Yaskawa INFORM job: X2_8B-21B(90,180)_REV_O.JBI

/JOB
//NAME X2_8B-21B(90,180)_REV_O
///FOLDERNAME X2
//POS
///NPOS 1154,1154,1154,53,0,0
///TOOL 0
///POSTYPE PULSE
///PULSE
C00000=-1415,-134459,-133802,-1969,12985,79332
C00001=-87080,-112473,-103627,-41798,51237,70410
C00002=-91681,-107347,-99471,-39221,49165,68848
C00003=-93439,-105106,-97054,-38371,48113,68361
C00004=-93441,-104864,-95967,-38672,47682,68565
C00005=-93504,-104969,-96260,-38564,47753,68495
C00006=-95585,-102642,-95415,-36914,47385,67494
C00007=-93504,-104969,-96260,-38564,47753,68495
C00008=-87147,-112175,-102116,-42180,50619,70689
C00009=-87145,-119394,-106475,-25944,48524,38750
C00010=-91166,-110510,-101811,-22693,48895,36705
C00011=-92650,-107060,-99920,-21494,49065,35962
C00012=-94767,-104655,-99060,-19829,49198,34943
C00013=-94484,-105085,-99259,-20052,49173,35080
C00014=-93721,-102513,-96995,-20598,49294,35408
C00015=-94484,-105085,-99259,-20052,49173,35080
C00016=-89209,-117497,-105909,-24366,48468,37757
C00017=-93166,-113214,-115710,-1969,57926,79332
C00018=-122366,-117496,-112293,16338,56235,67679
C00019=-123456,-103417,-106445,16337,59944,67813
C00020=-123456,-103539,-105172,16474,59132,67689
C00021=-123456,-103531,-105272,16463,59195,67698
C00022=-123128,-98284,-103303,16044,60561,68033
C00023=-123156,-99911,-105489,15984,61057,68095
C00024=-93710,-106990,-108704,-1652,56802,79139
C00025=-93766,-106412,-107148,-1629,56140,79127
C00026=-93768,-106433,-106329,-1638,55626,79135
C00027=-93918,-105383,-106173,-1535,56065,79069
C00028=-94164,-101296,-104676,-1361,57240,78956
C00029=-93895,-105502,-106499,-1547,56205,79076
C00030=-93151,-113316,-114305,-1998,57010,79354
C00031=-81072,-99391,-111155,-4750,63110,78553
C00032=-81984,-95120,-104767,-4287,61328,78293
C00033=-82103,-94682,-103397,-4241,60705,78273
C00034=-82106,-94924,-102383,-4271,59960,78300
C00035=-82089,-94934,-102578,-4276,60076,78302
C00036=-82803,-90374,-100753,-3806,61258,77993
C00037=-82089,-94934,-102578,-4276,60076,78302
C00038=-81057,-100006,-109908,-4804,62030,78604
C00039=-94004,-119945,-107122,49530,42714,48164
C00040=-93972,-116281,-97047,53343,39935,45878
C00041=-92833,-103149,-88492,51302,40218,47068
C00042=-93174,-100930,-87132,51219,40604,47120
C00043=-93174,-100493,-85792,51770,40220,46795
C00044=-93174,-101015,-87399,51095,40684,47186
C00045=-92955,-97894,-86230,50180,41136,47726
C00046=-93303,-100448,-87190,51023,40860,47230
C00047=-98055,-98607,-86499,53149,43882,46024
C00048=-96642,-96320,-85623,51883,43475,46780
C00049=-95342,-96864,-85830,51299,42647,47109
C00050=-97130,-98187,-86063,52744,43317,46271
C00051=-114545,-105110,-100746,39625,57097,48369
C00052=-113947,-102413,-97570,39574,56382,48359
C00053=-113947,-102278,-96691,39772,56015,48196
C00054=-113346,-99976,-96570,39024,56612,48763
C00055=-112899,-98120,-95866,38597,56823,49078
C00056=-114020,-99555,-96940,39169,57262,48705
C00057=-56302,-84822,-83054,-58022,66572,84014
C00058=-58361,-85953,-83540,-57558,65172,83717
C00059=-56302,-84822,-83054,-58022,66572,84014
C00060=-50122,-85714,-86741,-59061,71306,84454
C00061=-54195,-101901,-111197,-24063,62262,77343
C00062=-67243,-111926,-101536,21450,29925,69540
C00063=-66442,-101704,-94400,19916,30532,70304
C00064=-66308,-99858,-92576,19846,30336,70336
C00065=-66311,-99589,-91307,20230,29731,70137
C00066=-66308,-99960,-93112,19687,30597,70418
C00067=-70591,-100617,-92786,25268,31264,67678
C00068=-70591,-100325,-91437,25755,30647,67424
C00069=-68222,-99738,-91214,22742,30105,68906
C00070=-70591,-100606,-92729,25289,31242,67667
C00071=-66097,-110297,-96199,21577,27345,69446
C00072=-65719,-107666,-92844,21562,26575,69447
C00073=-65848,-106528,-92445,21497,26927,69482
C00074=-65365,-110699,-93884,21743,25627,69354
C00075=-67243,-111926,-101536,21450,29925,69540
C00076=-68963,-41843,-96211,-398,96948,-48811
C00077=-76932,-51697,-92360,2602,89609,-51106
C00078=-71886,-45093,-85416,705,88639,-49643
C00079=-71886,-45937,-84760,705,87803,-49648
C00080=-71886,-44632,-85753,705,89084,-49641
C00081=-68776,-90352,-95136,-4313,51281,-47645
C00082=-68803,-86754,-93636,-4241,52203,-47695
C00083=-68762,-92243,-95906,-4353,50785,-47617
C00084=-77446,-64871,-91176,8832,74282,-49527
C00085=-75907,-64612,-91046,8095,74185,-49034
C00086=-78150,-64967,-91224,9168,74335,-49752
C00087=-78150,-57569,-97635,8943,81990,-49191
C00088=-68963,-41843,-96211,-398,96948,-48811
C00089=-67385,-42511,-92598,-992,94393,-48367
C00090=-66773,-44328,-90253,-1220,92024,-48175
C00091=-66900,-44765,-89647,-1171,91425,-48205
C00092=-66773,-43962,-90441,-1221,92327,-48178
C00093=-69817,-49291,-93527,-72,91467,-49038
C00094=-102407,-61387,-79216,48101,75803,-74984
C00095=-99741,-62884,-79905,47237,74215,-74494
C00096=-102407,-61387,-79216,48101,75803,-74984
C00097=-71396,-101707,-96198,105,39560,-49678
C00098=-71544,-99303,-95354,247,40276,-49753
C00099=-71126,-105930,-97636,-165,38275,-49535
C00100=-74447,-120283,-111838,3099,39699,-51260
C00101=-57750,-84762,-113304,-22338,79933,-80646
C00102=-38298,-117376,-123136,-35520,84192,-83183
C00103=-31003,-114098,-105660,-45955,85390,-81321
C00104=-32496,-116782,-107403,-45795,84408,-81579
C00105=-34116,-118987,-108120,-45640,83088,-81742
C00106=-33779,-118873,-108083,-45678,83285,-81673
C00107=-33779,-118389,-106291,-45736,82677,-81394
C00108=-33116,-116007,-107005,-45711,84199,-81779
C00109=-43122,-77390,-91933,-43525,86904,-87571
C00110=-44353,-78017,-92219,-43231,86215,-87819
C00111=-45440,-79271,-92786,-42975,85486,-87990
C00112=-45102,-79332,-92813,-43057,85636,-87902
C00113=-45102,-79709,-91490,-43095,84888,-87585
C00114=-41853,-68825,-87871,-43817,88900,-87868
C00115=-48095,-31712,-66541,-47290,99218,-86920
C00116=-48762,-33638,-67810,-47108,98755,-86994
C00117=-49503,-35735,-69173,-46902,98237,-87073
C00118=-49389,-35416,-68966,-46933,98317,-87062
C00119=-49389,-36060,-68028,-46814,97684,-86756
C00120=-48487,-32850,-67294,-47182,98948,-86964
C00121=-45126,-25671,-76382,-49967,106798,-89554
C00122=-48508,-32956,-85951,-38791,109748,-85822
C00123=-73491,-115415,-129730,-12591,84406,-82629
C00124=-68604,-111632,-124361,34026,103601,-55041
C00125=-52690,-105642,-114364,31889,95098,-51390
C00126=-50963,-109289,-114635,31553,93010,-51314
C00127=-50968,-109442,-114037,31534,92627,-51422
C00128=-50963,-109237,-114816,31559,93129,-51281
C00129=-54701,-101748,-112541,32228,96580,-51739
C00130=-54580,-102143,-110625,32107,95358,-52042
C00131=-52710,-105778,-111943,31798,93771,-51772
C00132=-54580,-102143,-110625,32107,95358,-52042
C00133=-53574,-106836,-112314,31893,93817,-52092
C00134=-52008,-102475,-110737,31756,94333,-51344
C00135=-53574,-106836,-112314,31893,93817,-52092
C00136=-61074,-96775,-114868,33501,102293,-52496
C00137=-149084,-102156,-129577,22032,95315,-42360
C00138=-128569,-114069,-129208,14930,94899,-36248
C00139=-124702,-111484,-125119,14131,93099,-35189
C00140=-117407,-110681,-122838,12596,90996,-33018
C00141=-117407,-111232,-122133,12590,90297,-33088
C00142=-117407,-111153,-122240,12590,90402,-33077
C00143=-117516,-104258,-119840,12640,92435,-32906
C00144=-117407,-111153,-122240,12590,90402,-33077
C00145=-137517,-133828,-121685,31184,78220,-41365
C00146=-133868,-135584,-122192,30484,76378,-40422
C00147=-116503,-109521,-121739,12400,90787,-32743
C00148=-117639,-111560,-122305,12792,90174,-33159
C00149=-129920,-104375,-121589,15367,95339,-36612
C00150=-129920,-105073,-120932,15342,94602,-36705
C00151=-129920,-105823,-120129,15315,93754,-36812
C00152=-129920,-105714,-120250,15319,93879,-36798
C00153=-129568,-97895,-117405,15323,96007,-36416
C00154=-129817,-102709,-120162,15344,95301,-36587
C00155=-121595,-114825,-128025,13496,92670,-34216
C00156=-122629,-107467,-122921,17549,92277,-31147
C00157=-121348,-106187,-119304,17235,90519,-30969
C00158=-121348,-106897,-118296,17228,89578,-31103
C00159=-121348,-106810,-118429,17228,89701,-31085
C00160=-121327,-99353,-115727,17255,91773,-30786
C00161=-121340,-102686,-118046,17252,91502,-30828
C00162=-123984,-121300,-124584,22039,85383,-28695
C00163=-118596,-113071,-118409,20758,84424,-26972
C00164=-117828,-112575,-117002,20585,83663,-26833
C00165=-117596,-112721,-116348,20543,83158,-26838
C00166=-117643,-112201,-116474,20543,83493,-26797
C00167=-117846,-106122,-114344,20549,85245,-26570
C00168=-117643,-112201,-116474,20543,83493,-26797
C00169=-125192,-113488,-115877,22341,84450,-29296
C00170=-124919,-116220,-115928,22323,83104,-29449
C00171=-122352,-116155,-116251,21738,82647,-28614
C00172=-124919,-116220,-115928,22323,83104,-29449
C00173=-123984,-121300,-124584,22039,85383,-28695
C00174=-86442,-134681,-133724,-19248,79211,-32552
C00175=-86002,-121949,-124889,-19319,80358,-32581
C00176=-83173,-118115,-122503,-20102,81494,-31775
C00177=-83173,-118355,-121819,-20128,80982,-31690
C00178=-83173,-118313,-121945,-20123,81076,-31705
C00179=-84570,-111270,-119601,-19642,82802,-32476
C00180=-84061,-113318,-121554,-19798,83063,-32340
C00181=-99760,-154859,-112577,-64842,65446,-34340
C00182=-105860,-151698,-110493,-64559,61681,-35508
C00183=-106986,-150846,-109245,-64674,60811,-35545
C00184=-106922,-150967,-109400,-64661,60866,-35548
C00185=-107498,-146229,-108289,-63778,61296,-36463
C00186=-107239,-150553,-110467,-64221,61056,-36009
C00187=-103039,-154525,-109995,-65437,62710,-34223
C00188=-103986,-153521,-108660,-65576,61968,-34235
C00189=-103986,-153752,-108910,-65558,61982,-34250
C00190=-104831,-148338,-107690,-64592,62341,-35332
C00191=-104831,-154990,-115289,-64019,62915,-35911
C00192=-86002,-121949,-124889,-19319,80358,-32581
C00193=-89184,-120947,-124012,-18384,79622,-33578
C00194=-89184,-121311,-122777,-18433,78722,-33443
C00195=-89184,-121280,-122900,-18428,78809,-33455
C00196=-90163,-115208,-120930,-18039,80412,-34039
C00197=-89061,-121712,-124317,-18429,79452,-33511
C00198=-95932,-170316,-132534,-19010,48950,-33315
C00199=-95449,-171774,-131482,-19685,47748,-32835
C00200=-93413,-168537,-129826,-20545,48851,-32116
C00201=-93413,-168812,-130071,-20542,48860,-32116
C00202=-94803,-159418,-127836,-18887,51784,-33360
C00203=-94151,-164650,-129663,-19626,50457,-32799
C00204=-96358,-174071,-130551,-19748,45875,-32859
C00205=-95061,-171972,-129445,-20316,46563,-32383
C00206=-95061,-172212,-129646,-20316,46563,-32383
C00207=-96259,-163989,-127758,-18767,49173,-33508
C00208=-95716,-170264,-130833,-19432,48038,-33021
C00209=-120611,-122953,-119681,21560,80854,-22535
C00210=-120610,-122943,-118608,21593,80243,-22645
C00211=-120610,-122853,-116921,21650,79318,-22813
C00212=-120610,-122881,-117271,21638,79506,-22779
C00213=-120610,-122878,-117279,21638,79511,-22778
C00214=-120610,-122881,-117271,21638,79506,-22779
C00215=-120610,-122873,-117198,21640,79468,-22785
C00216=-120610,-122853,-117190,21640,79473,-22785
C00217=-120610,-122873,-117198,21640,79468,-22785
C00218=-120611,-122910,-120952,21522,81605,-22399
C00219=-86002,-120340,-127953,-19212,82925,-32989
C00220=-83173,-118115,-122503,-20102,81494,-31775
C00221=-83173,-118354,-121819,-20128,80983,-31690
C00222=-83173,-118313,-121945,-20123,81076,-31705
C00223=-84570,-111270,-119601,-19642,82802,-32476
C00224=-84061,-113318,-121554,-19798,83063,-32340
C00225=-99760,-154859,-112577,-64842,65446,-34340
C00226=-105859,-151698,-110493,-64559,61681,-35508
C00227=-106987,-150846,-109245,-64674,60811,-35545
C00228=-106922,-150967,-109400,-64660,60866,-35548
C00229=-107498,-146229,-108289,-63777,61296,-36463
C00230=-107240,-150553,-110467,-64221,61056,-36009
C00231=-103039,-154525,-109995,-65437,62710,-34223
C00232=-103986,-153521,-108660,-65576,61968,-34235
C00233=-103986,-153752,-108910,-65558,61982,-34249
C00234=-104831,-148338,-107690,-64592,62341,-35332
C00235=-104831,-154990,-115290,-64019,62915,-35911
C00236=-86002,-121950,-124889,-19319,80357,-32581
C00237=-89184,-120947,-124012,-18384,79622,-33578
C00238=-89184,-121311,-122777,-18433,78722,-33443
C00239=-89184,-121280,-122899,-18429,78809,-33455
C00240=-90163,-115207,-120930,-18039,80412,-34039
C00241=-89061,-121712,-124317,-18429,79452,-33511
C00242=-95932,-170316,-132534,-19010,48950,-33315
C00243=-95449,-171774,-131482,-19685,47748,-32835
C00244=-93413,-168536,-129826,-20544,48851,-32117
C00245=-93413,-168811,-130070,-20542,48860,-32116
C00246=-94803,-159417,-127836,-18887,51784,-33360
C00247=-94151,-164650,-129664,-19626,50457,-32799
C00248=-96358,-174071,-130551,-19748,45875,-32859
C00249=-95060,-171973,-129446,-20316,46563,-32383
C00250=-95061,-172212,-129646,-20316,46563,-32383
C00251=-96259,-163989,-127758,-18767,49173,-33508
C00252=-95716,-170264,-130834,-19432,48038,-33021
C00253=-120612,-120891,-127143,3106,87300,-4415
C00254=-120611,-122177,-124352,3111,84925,-4474
C00255=-120611,-122645,-122467,3116,83527,-4507
C00256=-120611,-122779,-121606,3119,82929,-4523
C00257=-120611,-122697,-122159,3117,83311,-4513
C00258=-120611,-122692,-122166,3117,83318,-4513
C00259=-120611,-122697,-122159,3117,83311,-4513
C00260=-120611,-121412,-126223,3107,86468,-4436
C00261=-120611,-118807,-129728,3107,89959,-4350
C00262=-120605,-132560,-136700,3104,87187,-4416
C00263=-53188,-122658,-121398,34453,103181,-41719
C00264=-53187,-122644,-116623,34032,100735,-42492
C00265=-53184,-122447,-115007,33919,99986,-42724
C00266=-53180,-122268,-113886,33849,99484,-42877
C00267=-53186,-122531,-115629,33961,100272,-42636
C00268=-53233,-122033,-113114,32057,113501,-44659
C00269=-53229,-122037,-113108,32057,113495,-44659
C00270=-53233,-122033,-113114,32057,113501,-44659
C00271=-53127,-122157,-112856,34567,84618,-41563
C00272=-53132,-122146,-112848,34568,84621,-41564
C00273=-53127,-122157,-112856,34567,84618,-41563
C00274=-53124,-122720,-116247,34514,86111,-41098
C00275=-61684,-126457,-131749,21672,103686,-55019
C00276=-68676,-133744,-131015,10578,108811,-68614
C00277=-80160,-118182,-130261,-41,125141,-81817
C00278=-80187,-122370,-123619,-70,118933,-81856
C00279=-80183,-122639,-122398,-68,118043,-81854
C00280=-80181,-122756,-121636,-67,117515,-81853
C00281=-80184,-122603,-122588,-68,118179,-81854
C00282=-80182,-122615,-122584,-67,118170,-81853
C00283=-80184,-122603,-122588,-68,118179,-81854
C00284=-80200,-121154,-126606,-75,121396,-81862
C00285=-109164,-117358,-132635,-7350,119146,-48306
C00286=-144183,-119511,-130571,-15498,107286,-7245
C00287=-197934,-122815,-127402,-28006,89082,55776
C00288=-202772,-123889,-124791,-27048,85608,54814
C00289=-204705,-124106,-122314,-26692,83530,54575
C00290=-204705,-124189,-120905,-26732,82711,54762
C00291=-205113,-122699,-120601,-26621,83104,54520
C00292=-208506,-122040,-120392,-25870,82241,53457
C00293=-204510,-125657,-121990,-26775,82699,54838
C00294=-204510,-125393,-124777,-26704,84359,54459
C00295=-217123,-144581,-130617,-26990,80795,43719
C00296=-208514,-157553,-136215,-22784,79668,13108
C00297=-208134,-153606,-128050,-23049,77001,13769
C00298=-209226,-147410,-126429,-22728,78719,13024
C00299=-208514,-151468,-127497,-22936,77598,13510
C00300=-218941,-132344,-125800,-20692,83017,8703
C00301=-218940,-132255,-124809,-20728,82492,8794
C00302=-218940,-132304,-125288,-20718,82746,8752
C00303=-219615,-126196,-123449,-20528,84462,8218
C00304=-218940,-132304,-125288,-20718,82746,8752
C00305=-200084,-117243,-114643,-37064,92847,22860
C00306=-201812,-115748,-114150,-36926,92488,22266
C00307=-218940,-132304,-125288,-20718,82746,8752
C00308=-203904,-153254,-131986,6783,67239,16317
C00309=-203904,-152472,-130784,6798,66902,16298
C00310=-203904,-152823,-131321,6790,67052,16308
C00311=-205098,-146177,-129554,7075,69466,16016
C00312=-203904,-152823,-131321,6790,67052,16308
C00313=-223566,-125183,-123361,20045,84784,-13848
C00314=-220870,-123350,-122791,19484,84702,-12913
C00315=-222373,-123821,-125769,19771,86556,-13139
C00316=-208514,-151468,-127497,-22936,77598,13510
C00317=-208514,-156517,-134755,-22805,79329,13174
C00318=-197934,-122815,-127402,-28006,89082,55776
C00319=-202772,-123889,-124791,-27048,85608,54814
C00320=-204705,-124106,-122314,-26692,83530,54575
C00321=-204705,-124189,-120905,-26732,82711,54762
C00322=-205113,-122699,-120601,-26621,83104,54520
C00323=-208506,-122040,-120392,-25870,82241,53457
C00324=-204510,-125657,-121990,-26775,82699,54838
C00325=-204510,-125393,-124777,-26704,84359,54459
C00326=-217123,-144581,-130617,-26990,80795,43719
C00327=-216657,-144339,-132121,-20327,83655,24427
C00328=-208514,-151468,-127497,-22936,77598,13510
C00329=-209226,-147410,-126429,-22728,78719,13024
C00330=-208514,-151468,-127497,-22936,77598,13510
C00331=-208514,-156517,-134755,-22805,79329,13174
C00332=-187736,-116553,-120968,-36188,98329,31010
C00333=-144869,-104708,-130913,697,92502,-12445
C00334=-97478,-100538,-119508,25976,122096,-72949
C00335=-94415,-115583,-120723,24602,114867,-73486
C00336=-94145,-116737,-119872,24403,113768,-73630
C00337=-94090,-116915,-118863,24267,113100,-73760
C00338=-94227,-118887,-121662,24392,113788,-73658
C00339=-94618,-126072,-123928,23885,111795,-74261
C00340=-93811,-121058,-122280,24303,112998,-73673
C00341=-123165,-134656,-120887,30393,109989,-65140
C00342=-122877,-135920,-118822,30065,108215,-65520
C00343=-120918,-135771,-118381,30417,107339,-64954
C00344=-122877,-135920,-118822,30065,108215,-65520
C00345=-123434,-129548,-123417,31323,113703,-64157
C00346=-83798,-143971,-127552,34208,94145,-53659
C00347=-12921,-128304,-123041,22509,73309,-31557
C00348=-1276,-141206,-132907,9958,77401,-32714
C00349=458,-143834,-132257,9551,75469,-32266
C00350=455,-143428,-130846,9594,74819,-32314
C00351=455,-143488,-131041,9589,74909,-32308
C00352=3648,-143226,-130969,8703,74636,-31209
C00353=1152,-143828,-132318,9375,75428,-32023
C00354=8026,-156372,-135202,7630,70086,-29960
C00355=9901,-151141,-133831,7007,71746,-29188
C00356=9901,-150525,-132660,7023,71345,-29214
C00357=9901,-150622,-132845,7021,71407,-29209
C00358=13681,-148784,-132355,5888,71743,-27846
C00359=12497,-150457,-134690,6220,72408,-28233
C00360=-126606,-101457,-128935,16844,101795,-36174
C00361=-152779,-135138,-131563,2515,76140,-19155
C00362=-150820,-122490,-124749,1875,78392,-18455
C00363=-150097,-118368,-121531,1645,78513,-18212
C00364=-150095,-118599,-120646,1648,77850,-18220
C00365=-147666,-112236,-119185,871,80184,-17389
C00366=-146670,-110099,-118456,556,80825,-17059
C00367=-148658,-114325,-119887,1186,79554,-17722
C00368=-87079,-91764,-103818,-42328,107533,9448
C00369=-87027,-91004,-101788,-42122,106912,9740
C00370=-89264,-90509,-101588,-42089,105978,9119
C00371=-87027,-91004,-101788,-42122,106912,9740
C00372=-87391,-90282,-107909,-43186,109836,8282
C00373=-92115,-87061,-118989,-19004,94950,-3823
C00374=-109005,-100727,-117090,5533,93286,-3886
C00375=-109005,-102030,-115406,5521,91587,-3960
C00376=-109005,-101552,-116078,5524,92244,-3931
C00377=-107643,-92243,-112443,5266,94693,-3390
C00378=-109005,-99994,-117863,5541,94135,-3847
C00379=-92115,-87061,-118989,-19004,94950,-3823
C00380=-78975,-130870,-123203,19746,71053,-12291
C00381=-74317,-97013,-111518,17407,83606,-9286
C00382=-74211,-95430,-110119,17377,83539,-9259
C00383=-74211,-95892,-109317,17397,82840,-9358
C00384=-75305,-113551,-114600,17838,69768,-10493
C00385=-78326,-111051,-111958,19079,70114,-11550
C00386=-78379,-106110,-110225,18937,71523,-11339
C00387=-78263,-116865,-113913,19272,68408,-11810
C00388=-85880,-113569,-112821,22054,71256,-14152
C00389=-85920,-114580,-110580,22309,69503,-14507
C00390=-82054,-114988,-110714,20879,68380,-13249
C00391=-85920,-114580,-110580,22309,69503,-14507
C00392=-78975,-130870,-123203,19746,67177,-12291
C00393=-159950,-115131,-126913,-23322,109234,64770
C00394=-163413,-124246,-126581,-22686,103792,64589
C00395=-164859,-127477,-125491,-22457,101245,64551
C00396=-164857,-127553,-124648,-22406,100728,64651
C00397=-164862,-127370,-126252,-22506,101730,64457
C00398=-158275,-145382,-129341,-21795,96649,67831
C00399=-159759,-153222,-131425,-21726,93697,67826
C00400=-158275,-145382,-129341,-21795,96649,67831
C00401=-157577,-144643,-126617,-21696,95625,68274
C00402=-160219,-140867,-125578,-21868,96138,67212
C00403=-157577,-144643,-126617,-21696,95625,68274
C00404=-152631,-134238,-128202,-21932,102817,68768
C00405=-146941,-123801,-133763,-3444,102850,52685
C00406=-136178,-116173,-124987,31736,84906,22811
C00407=-134413,-106132,-117362,31242,84680,23412
C00408=-134231,-105594,-115694,31219,83968,23286
C00409=-134230,-105863,-115134,31239,83552,23172
C00410=-134007,-104199,-114803,31151,84035,23389
C00411=-133473,-100630,-113499,30965,84737,23780
C00412=-134315,-106237,-115533,31260,83629,23161
C00413=-136272,-117460,-124003,31807,83855,22481
C00414=-136226,-116324,-125056,31750,84893,22789
C00415=-134474,-106353,-117504,31259,84679,23389
C00416=-134275,-105758,-115681,31235,83904,23252
C00417=-134274,-105987,-115198,31252,83547,23154
C00418=-134027,-104733,-115029,31162,83924,23350
C00419=-133465,-100971,-113658,30966,84667,23763
C00420=-134308,-106598,-115693,31262,83551,23142
C00421=-178993,-121773,-123174,38769,99022,10273
C00422=-175539,-115427,-119854,38657,98481,11541
C00423=-175539,-115857,-118311,38525,97555,11203
C00424=-175539,-115829,-118427,38535,97623,11227
C00425=-173168,-111114,-116839,38478,97741,12267
C00426=-174072,-113112,-119760,38657,98741,12252
C00427=-136269,-117902,-124178,31812,83752,22453
C00428=-139753,-124875,-130430,383,75663,-26245
C00429=-143223,-157944,-133481,-5653,58679,-38405
C00430=-140983,-144085,-126452,-6488,61628,-37698
C00431=-140148,-138933,-122655,-6835,62006,-37402
C00432=-140147,-138616,-121921,-6853,61719,-37384
C00433=-140691,-136506,-121897,-6553,62737,-37651
C00434=-138669,-131542,-120459,-7325,64564,-37004
C00435=-140691,-136506,-121897,-6553,62737,-37651
C00436=-145148,-139028,-124584,-4588,62787,-39337
C00437=-159973,-92454,-110285,14523,90938,-48717
C00438=-158765,-97223,-112137,14224,89465,-48492
C00439=-159973,-92454,-110285,14523,90938,-48717
C00440=-164681,-91509,-114703,15696,94847,-49769
C00441=-142525,-105883,-132766,-7713,103357,-60336
C00442=-90751,-115691,-121566,-36045,104861,-61043
C00443=-92920,-122587,-117773,-35137,99152,-60047
C00444=-93124,-123070,-117553,-35091,98753,-60003
C00445=-93124,-123008,-116878,-35050,98435,-59900
C00446=-93160,-123063,-117190,-35068,98555,-59953
C00447=-95752,-125144,-117838,-34977,96947,-60505
C00448=-93160,-123063,-117190,-35068,98555,-59953
C00449=-92038,-109836,-114685,-38536,89453,-57060
C00450=-86810,-100893,-104585,-47463,92019,-56975
C00451=-88449,-102594,-103600,-47188,90148,-56855
C00452=-88449,-102618,-102426,-47172,89639,-56610
C00453=-88449,-102603,-103366,-47184,90046,-56806
C00454=-85133,-99388,-102162,-47637,92393,-56350
C00455=-85168,-99488,-101153,-47595,91912,-56132
C00456=-86978,-101259,-101820,-47360,90627,-56378
C00457=-84037,-98201,-102123,-47804,93363,-56297
C00458=-108771,-112096,-123986,-16313,85813,-59347
C00459=-109769,-112695,-132242,-3132,99947,-61138
C00460=-127404,-127157,-120795,27540,73197,-60883
C00461=-120526,-123085,-115007,25540,69700,-59025
C00462=-119461,-122312,-114032,25210,69192,-58723
C00463=-119461,-122116,-113003,25293,68708,-58832
C00464=-119461,-122312,-114032,25210,69192,-58723
C00465=-94655,-112249,-115827,-1041,75214,-51009
C00466=-93364,-111129,-115444,-1499,75574,-50577
C00467=-121213,-123445,-114215,25873,69302,-59387
C00468=-127714,-127278,-119628,27738,72603,-61150
C00469=-140848,-129628,-128054,17424,84805,-27418
C00470=-127903,-106251,-120637,17388,91568,-15860
C00471=-124887,-98361,-114445,16717,91208,-14907
C00472=-124532,-94860,-112080,16625,91471,-14753
C00473=-117832,-103976,-115449,15062,87719,-13014
C00474=-118209,-109888,-118953,15141,86934,-13233
C00475=-120968,-118649,-124805,15800,86569,-14208
C00476=-112726,-101228,-128594,1890,90279,15897
C00477=-102865,-105549,-130121,-1361,88970,18873
C00478=-85416,-143080,-122146,-23399,58401,32529
C00479=-89847,-131888,-116792,-20882,59491,30436
C00480=-92125,-126361,-114096,-19602,60042,29398
C00481=-92108,-126361,-114086,-19611,60041,29405
C00482=-94963,-119193,-112807,-13876,65309,25883
C00483=-99230,-109273,-111594,-7832,72910,21884
C00484=-97558,-114678,-114533,-8498,72116,22521
C00485=-94805,-124749,-120489,-9597,70928,23580
C00486=-89899,-115674,-129227,-15589,81503,27304
C00487=-94000,-113154,-130859,1035,116659,-75004
C00488=-93721,-118000,-129934,5060,122177,-74127
C00489=-93715,-120352,-127357,4900,119392,-74256
C00490=-95346,-120435,-125547,4467,118331,-74923
C00491=-87734,-123112,-126247,6115,116903,-72103
C00492=-93725,-120284,-127319,4898,119404,-74259
C00493=-93731,-117931,-129895,5059,122189,-74130
C00494=-92605,-107385,-114202,-42080,118626,-78084
C00495=-94957,-117308,-114744,-40643,113912,-77125
C00496=-96859,-119647,-113709,-40343,111617,-77062
C00497=-96820,-119688,-113698,-40330,111613,-77042
C00498=-92369,-120637,-111842,-39132,112371,-75247
C00499=-87506,-133441,-114197,-38673,106213,-75021
C00500=-90618,-118755,-112828,-39302,114392,-75239
C00501=-88476,-109244,-112462,-40625,118981,-76164
C00502=-73726,-95231,-122050,-23824,117115,-78775
C00503=-68964,-113071,-130294,19412,109419,-80322
C00504=-55630,-112625,-122011,35520,97927,-81697
C00505=-52390,-118820,-120628,34805,93310,-81881
C00506=-53603,-103093,-112884,36459,100480,-79984
C00507=-59619,-117562,-114740,37336,94951,-84077
C00508=-56690,-122472,-119439,35129,92879,-83747
C00509=-59872,-116629,-120975,35716,97415,-83571
C00510=-61517,-148095,-119735,48293,75564,-80066
C00511=-55473,-148057,-116974,48060,71191,-79214
C00512=-53771,-146175,-114985,47935,70110,-78894
C00513=-54494,-144748,-112549,48210,69974,-79344
C00514=-55476,-147094,-115701,48129,70996,-79318
C00515=-61520,-147186,-118480,48348,75358,-80173
C00516=-87978,-108563,-128727,6750,125872,-71649
C00517=-93715,-120352,-127357,4900,119392,-74256
C00518=-94748,-123674,-126724,4558,117361,-74733
C00519=-87347,-125535,-127084,6155,116151,-72000
C00520=-93725,-120284,-127319,4898,119404,-74259
C00521=-93731,-117931,-129895,5059,122189,-74130
C00522=-92605,-107385,-114202,-42080,118626,-78084
C00523=-94957,-117308,-114744,-40643,113912,-77125
C00524=-96514,-122009,-114462,-40074,111194,-76723
C00525=-96015,-122145,-114253,-39942,111269,-76518
C00526=-92174,-122830,-112540,-38890,111906,-74970
C00527=-86945,-136787,-114983,-38317,105485,-74493
C00528=-90618,-118755,-112828,-39302,114392,-75239
C00529=-88476,-109244,-112462,-40625,118981,-76164
C00530=-73726,-95231,-122050,-23824,117115,-78775
C00531=-68964,-113071,-130294,19412,109419,-80322
C00532=-55630,-112625,-122011,35520,97927,-81697
C00533=-52390,-118820,-120628,34805,93310,-81881
C00534=-47304,-107066,-116669,31636,98225,-78870
C00535=-58547,-113359,-113266,37552,97245,-82829
C00536=-56690,-122472,-119439,35129,92879,-83747
C00537=-59872,-116629,-120975,35716,97415,-83571
C00538=-61517,-148095,-119735,48293,75564,-80066
C00539=-55473,-148057,-116974,48060,71191,-79214
C00540=-53043,-147267,-115261,47953,69457,-78858
C00541=-53748,-146178,-113424,48182,69442,-79233
C00542=-55476,-147094,-115701,48129,70996,-79318
C00543=-61520,-147186,-118480,48348,75358,-80173
C00544=-69196,-132761,-125763,48066,87564,-77891
C00545=-67178,-112107,-133350,-9560,121946,-71499
C00546=-53652,-115588,-130730,-10921,119132,-80041
C00547=-53631,-118653,-128170,-10572,116038,-79726
C00548=-49406,-128725,-131842,-9345,109854,-77674
C00549=-50301,-131456,-131647,-9328,108248,-77863
C00550=-56808,-119713,-126858,-10890,114305,-80736
C00551=-54286,-118284,-126258,-10586,114987,-79865
C00552=-57104,-120165,-127558,-2939,114426,-79867
C00553=-59155,-122085,-128309,860,113653,-80114
C00554=-38667,-169406,-136982,4491,100158,-73221
C00555=-53493,-120154,-126714,1639,113579,-78070
C00556=-53512,-117734,-129516,1682,116546,-78033
C00557=-64263,-112177,-127274,18013,116425,-52133
C00558=-53349,-113292,-116223,34708,105130,-41711
C00559=-53347,-113647,-113946,34435,103813,-42137
C00560=-52680,-112871,-112467,34368,103124,-42082
C00561=-58031,-122280,-112065,36284,98076,-45699
C00562=-53343,-113729,-112902,34324,103242,-42318
C00563=-53345,-113489,-115217,34581,104530,-41905
C00564=-83368,-135406,-127982,43757,111124,24122
C00565=-107112,-148704,-121184,48737,110155,73723
C00566=-107085,-142005,-111593,48000,108472,72828
C00567=-107084,-140010,-108705,47787,107957,72557
C00568=-87331,-137626,-115833,38185,104318,80918
C00569=-107136,-152953,-127712,-1089,113260,57660
C00570=-107220,-158026,-128566,-1900,111074,56787
C00571=-107059,-148801,-134211,-1989,119286,56706
C00572=-109333,-147161,-118098,47834,110594,72761
C00573=-109333,-141938,-110765,47268,109335,72096
C00574=-106839,-147244,-109723,47050,105697,71521
C00575=-96955,-158208,-128899,-2670,111185,56030
C00576=-107130,-144670,-115956,-40497,90070,47196
C00577=-107133,-145289,-116877,-40503,90261,47122
C00578=-107139,-146938,-119316,-40521,90762,46927
C00579=-81304,-146505,-131302,-46256,99624,33732
C00580=-42290,-135810,-134986,-6789,56953,-43412
C00581=-53482,-111499,-99357,-5283,31563,-44884
C00582=-53488,-110753,-96932,-5448,30458,-44798
C00583=-53106,-110845,-96482,-5998,30161,-44520
C00584=-53143,-110117,-93832,-6189,28906,-44421
C00585=-53188,-109818,-93168,-6175,28651,-44427
C00586=-53095,-108922,-90553,-6542,27518,-44240
C00587=-53472,-108968,-91791,-5862,28222,-44586
C00588=-53466,-109889,-94290,-5675,29282,-44681
C00589=-93748,-113667,-111432,27227,62688,-41579
C00590=-93751,-113561,-109328,27520,61581,-41869
C00591=-94535,-110348,-107800,27711,62471,-41963
C00592=-94560,-109570,-102150,28499,59749,-42715
C00593=-93743,-112935,-104615,28181,59286,-42489
C00594=-93741,-113330,-106821,27872,60309,-42206
C00595=-53707,-103235,-126817,-3349,90409,-72793
C00596=-53694,-107630,-124107,-3352,86490,-72685
C00597=-53689,-108955,-122884,-3357,85060,-72645
C00598=-53697,-108940,-122873,-3354,85062,-72648
C00599=-53721,-108898,-122839,-3346,85062,-72656
C00600=-53729,-108884,-122827,-3345,85059,-72658
C00601=-53735,-107561,-124050,-3339,86489,-72698
C00602=-53748,-103173,-126762,-3336,90406,-72805
C00603=-44251,-68518,-112793,-6305,100072,-70363
C00604=-80270,30794,-42629,-11133,115571,-76543
C00605=-69737,67118,16632,-42575,112328,-80617
C00606=-69636,63823,22197,-49512,110599,-81416
C00607=-67564,55530,12856,-50142,112647,-81508
C00608=-66424,44944,1253,-49852,108764,-84350
C00609=-65618,29495,-14632,-48008,102670,-88237
C00610=-64581,15750,-27557,-48396,103780,-88326
C00611=-64160,11595,-31362,-48525,104124,-88308
C00612=-61878,-10748,-50140,-48981,105285,-87846
C00613=-62672,195,-41330,-51307,112408,-84907
C00614=-58944,10301,-35991,-52571,115494,-84879
C00615=-69716,-6230,-69222,-29298,97742,-75748
C00616=-102330,-22799,-82036,11222,88832,-73278
C00617=-48313,-118911,-129560,19207,92704,-27073
C00618=-53495,-110604,-121584,20154,93282,-28749
C00619=-53400,-112789,-120712,20093,91701,-28982
C00620=-53738,-109625,-119688,20178,92712,-28930
C00621=-53963,-109991,-119979,20218,92760,-28997
C00622=-54259,-112639,-122766,20278,93161,-29031
C00623=-53522,-108468,-123882,20258,95652,-28360
C00624=-66910,-101677,-117691,1645,82254,17515
C00625=-66905,-103395,-115374,1652,79946,17486
C00626=-66559,-103296,-114213,1536,79276,17588
C00627=-66525,-103141,-114029,1523,79241,17602
C00628=-67620,-103650,-114144,1902,79074,17240
C00629=-69968,-104694,-109483,10896,71665,17276
C00630=-74363,-105584,-109420,12680,71802,15748
C00631=-66783,-105788,-110032,11324,70201,18483
C00632=-66785,-105108,-112553,11207,72068,18659
C00633=-34610,-119076,-126707,-31995,89279,47352
C00634=-26693,-119602,-105841,-51320,82883,62074
C00635=-26676,-118953,-103885,-51392,82336,62389
C00636=-26611,-118260,-103653,-51381,82509,62328
C00637=-26639,-116853,-99731,-51529,81413,62927
C00638=-26666,-118021,-101324,-51491,81640,62785
C00639=-26683,-118745,-103309,-51412,82173,62476
C00640=-26741,-121947,-116429,-51038,86269,60171
C00641=-80158,-111738,-121779,-46707,81282,-33331
C00642=-80124,-114295,-114082,-47454,77096,-31277
C00643=-80115,-114367,-110881,-47781,75720,-30584
C00644=-79768,-115533,-110081,-48056,75157,-30124
C00645=-79863,-115342,-112075,-47802,76014,-30606
C00646=-81971,-122337,-112055,-47997,72434,-29847
C00647=-79704,-115764,-110171,-48082,75146,-30085
C00648=-122148,-120937,-111499,-32844,53810,-41506
C00649=-126062,-118880,-110838,-30416,52910,-43086
C00650=-126117,-120875,-113087,-30250,53200,-43207
C00651=-80061,-114542,-114188,-47480,77086,-31241
C00652=-80063,-113108,-120040,-30435,104055,-77976
C00653=-80050,-114212,-116860,-30086,101864,-77373
C00654=-80380,-112077,-114717,-30053,101557,-77419
C00655=-79932,-114590,-112006,-35005,85347,-77215
C00656=-79912,-114566,-112044,-35008,85386,-77219
C00657=-80479,-112475,-109427,-36632,80098,-77307
C00658=-80029,-114714,-111597,-36713,80437,-77233
C00659=-82440,-93132,-104306,-35744,84828,-79668
C00660=-83378,-90315,-100640,-35536,83784,-79702
C00661=-86724,-76310,-94495,-34501,85296,-81493
C00662=-81341,-82881,-101909,-35963,88366,-80388
C00663=-80042,-114535,-115070,-36542,82240,-77847
C00664=-80040,-111621,-122742,-8414,85267,-41918
C00665=-80035,-113457,-119567,-8450,82400,-41723
C00666=-81798,-124774,-120168,-7328,73182,-41674
C00667=-80327,-109577,-118133,2572,87034,-53415
C00668=-79380,-112621,-119090,2349,86031,-53125
C00669=-78889,-114029,-118891,6085,83597,-58153
C00670=-80002,-113603,-119620,10752,83390,-63441
C00671=-80006,-103113,-128729,10775,94202,-62513
C00672=-39776,-103787,-110683,-21075,62663,59255
C00673=-39766,-104399,-107995,-21452,60825,59622
C00674=-43409,-99604,-106611,-16852,63393,58055
C00675=-40129,-102322,-105584,-21337,60345,59571
C00676=-43388,-110191,-108436,-20000,57391,58823
C00677=-43700,-110741,-108624,-19856,57161,58737
C00678=-39744,-104425,-108009,-21464,60826,59630
C00679=-39754,-103814,-110697,-21087,62664,59263
C00680=-47977,-106691,-119962,-23629,83327,62671
C00681=-66867,-99660,-121232,-22132,99220,62132
C00682=-66851,-102572,-118810,-21937,96446,62653
C00683=-76349,-133711,-127427,-14100,78462,52804
C00684=-72951,-136123,-126583,-15051,77356,54134
C00685=-69979,-137998,-126184,-15851,76755,55266
C00686=-66851,-103895,-117201,-21852,94891,62938
C00687=-66868,-101493,-119792,-22004,97521,62449
C00688=-74321,-107832,-126985,11736,80239,61811
C00689=-66584,-114412,-108983,34198,49386,64476
C00690=-66581,-113854,-105403,35147,47795,63826
C00691=-60579,-124686,-103463,33716,33360,60449
C00692=-66753,-108025,-100247,35350,47717,63701
C00693=-67225,-112450,-100574,36771,46222,62781
C00694=-66567,-113311,-102857,35821,46729,63375
C00695=-66569,-114089,-106515,34851,48256,64025
C00696=-52763,-107501,-118592,5184,62268,61653
C00697=-39766,-104399,-107995,-21452,60825,59622
C00698=-41836,-96032,-105143,-17549,64604,58460
C00699=-42867,-98847,-106225,-17119,63645,58220
C00700=-46364,-107274,-109273,-15652,60551,57331
C00701=-47095,-108712,-109781,-15314,60002,57124
C00702=-39744,-104425,-108009,-21464,60826,59630
C00703=-39754,-103814,-110697,-21087,62664,59263
C00704=-47977,-106691,-119962,-23629,83327,62671
C00705=-66867,-99660,-121232,-22132,99220,62132
C00706=-66851,-102572,-118810,-21937,96446,62653
C00707=-73941,-131664,-126990,-14688,79641,53509
C00708=-72144,-132205,-126529,-15161,79422,54161
C00709=-66827,-135529,-125774,-16544,78356,56172
C00710=-66851,-103895,-117201,-21852,94891,62938
C00711=-66868,-101493,-119792,-22004,97521,62449
C00712=-74321,-107832,-126985,11736,80239,61811
C00713=-66584,-114412,-108983,34198,49386,64476
C00714=-66581,-113854,-105403,35147,47795,63826
C00715=-58452,-122882,-102720,31277,32940,61754
C00716=-58418,-124907,-102492,32276,32098,61343
C00717=-58598,-129664,-102309,34863,30024,60018
C00718=-66567,-113311,-102857,35821,46729,63375
C00719=-66569,-114089,-106515,34851,48256,64025
C00720=-66614,-114312,-115902,32344,53032,65825
C00721=-26293,-124733,-123676,35115,86081,77095
C00722=-26278,-124914,-120130,35186,84196,76502
C00723=-26550,-125631,-118910,35285,83385,76132
C00724=-26140,-123752,-118256,35186,83681,76394
C00725=-26301,-124893,-120124,35190,84211,76498
C00726=-26317,-124710,-123669,35119,86096,77090
C00727=-26368,-124828,-121889,39154,95960,78120
C00728=-26350,-124746,-118556,38992,94373,77544
C00729=-26342,-124553,-116950,38932,93670,77290
C00730=-26340,-123995,-113991,38847,92461,76851
C00731=-26347,-124286,-115407,38884,93032,77056
C00732=-26365,-124761,-118865,39006,94524,77592
C00733=-26264,-124528,-116402,47920,86072,68134
C00734=-26249,-123768,-112787,47988,84810,67516
C00735=-26243,-123374,-111311,48022,84325,67278
C00736=-26226,-122772,-109280,48074,83674,66962
C00737=-26232,-123227,-110778,48035,84146,67194
C00738=-26247,-124165,-114452,47952,85370,67795
C00739=-82585,-123093,-118421,52491,64599,59558
C00740=-107155,-118824,-102398,58122,50036,52281
C00741=-107155,-117467,-98958,59145,49269,51564
C00742=-97769,-115596,-103462,42332,48327,50952
C00743=-106191,-118370,-109045,10471,43744,62968
C00744=-106214,-118343,-108967,10497,43713,62952
C00745=-107926,-118894,-109147,11962,43778,62125
C00746=-109818,-119504,-109023,13611,43678,61235
C00747=-128826,-124074,-107976,29086,45857,52131
C00748=-107169,-120346,-107141,7797,39493,71540
C00749=-108433,-119625,-117514,7930,46308,71537
C00750=-107111,-122100,-111275,39348,45202,56077
C00751=-107109,-117760,-98763,43179,41028,53713
C00752=-107213,-117629,-97756,43683,40670,53413
C00753=-106421,-119420,-102480,12268,36878,61896
C00754=-109448,-120604,-102361,14254,36543,60803
C00755=-88192,-110716,-101036,-23203,47482,70245
C00756=-83847,-106333,-107319,-25140,55050,70229
C00757=-110745,-121766,-106380,43469,44759,53583
C00758=-110745,-121766,-106380,43469,44759,53584
C00759=-120731,-110814,-96413,59684,53172,46713
C00760=-94986,-115649,-101302,-12294,38121,75258
C00761=-110957,-117259,-94521,-45268,37979,76630
C00762=-107127,-114270,-91297,-56630,43098,80056
C00763=-102543,-110504,-99650,-53136,49996,77723
C00764=-93612,-109275,-133010,12113,75674,64968
C00765=-74458,-81913,-116300,25886,107898,47202
C00766=-74285,-84923,-113224,25351,104735,46539
C00767=-74085,-86300,-112083,25142,103399,46313
C00768=-71499,-76504,-108067,25490,106819,45523
C00769=-62961,-60085,-100217,24652,107848,48688
C00770=-60437,-59805,-99888,23461,105440,51393
C00771=-60588,-58283,-100875,23679,106756,51616
C00772=-60637,-54628,-103477,24231,109960,52288
C00773=-76657,-70403,-83915,51355,64349,40407
C00774=-74830,-68241,-74355,53953,55282,38932
C00775=-73110,-62379,-68708,53436,54020,39148
C00776=-73182,-62563,-68609,53555,53963,39058
C00777=-36930,-67607,-75173,-26029,44061,77403
C00778=-80523,-89058,-85253,18218,36719,55154
C00779=-82272,-90569,-85112,18702,34759,56728
C00780=-81508,-95500,-88175,18158,33969,56993
C00781=-81043,-103588,-94156,17854,33413,57140
C00782=-82846,-88179,-88219,41798,48730,43563
C00783=-81818,-81213,-82326,41198,48211,43888
C00784=-79663,-80074,-80946,37957,46333,45127
C00785=-64011,-84834,-85332,4259,39755,58703
C00786=-75846,-87347,-86370,15921,40584,52659
C00787=-47572,-67654,-78731,-37306,60592,66422
C00788=-46339,-68382,-80235,-37741,61555,66618
C00789=-42699,-70655,-83815,-39176,63943,67342
C00790=-43803,-67144,-92021,-36183,69839,64523
C00791=-86906,-70734,-117845,25978,101850,24881
C00792=-194376,-118372,-116958,36622,58194,-75254
C00793=-187943,-106127,-101715,33777,52366,-74665
C00794=-187951,-105693,-98645,34509,50978,-75202
C00795=-187954,-105458,-97394,34809,50440,-75417
C00796=-187960,-105469,-97402,34805,50444,-75420
C00797=-187927,-105629,-98482,19599,46235,-60273
C00798=-187923,-105820,-99644,19403,46817,-60144
C00799=-187914,-106157,-102495,18928,48312,-59826
C00800=-188021,-109107,-91072,54887,40419,-77132
C00801=-188025,-108188,-88773,55807,39869,-77674
C00802=-188027,-107805,-87846,56180,39654,-77892
C00803=-188036,-107761,-87717,56242,39627,-77928
C00804=-188035,-108145,-88644,55869,39841,-77710
C00805=-188030,-109068,-90945,54948,40390,-77168
C00806=-188015,-114130,-110744,41340,72657,-75143
C00807=-188018,-113864,-107763,41683,71368,-75679
C00808=-188019,-113684,-106544,41824,70871,-75888
C00809=-188009,-113674,-106577,41816,70886,-75877
C00810=-188008,-113852,-107795,41674,71383,-75668
C00811=-188005,-114114,-110775,41332,72673,-75132
C00812=-187933,-113872,-110928,18210,58720,-57176
C00813=-187882,-113256,-105308,-719,43762,-42538
C00814=-187896,-112711,-102669,-725,42418,-42533
C00815=-187852,-113170,-101841,-775,41671,-42505
C00816=-187778,-112374,-98354,-1639,37547,-42296
C00817=-187899,-111729,-99017,-1491,38283,-42378
C00818=-187886,-112431,-101600,-1465,39511,-42393
C00819=-192869,-127835,-120494,22551,66263,-53872
C00820=-188079,-122619,-114609,40714,83609,-61664
C00821=-188077,-122103,-112045,40794,82601,-62056
C00822=-188097,-121812,-110726,41966,87288,-59780
C00823=-188097,-121769,-110559,41966,87227,-59806
C00824=-188105,-121282,-108770,41980,86589,-60067
C00825=-188106,-121566,-109755,41972,86936,-59927
C00826=-188110,-122188,-112187,41960,87826,-59570
C00827=-188058,-121965,-125191,40549,88870,-59628
C00828=-104402,-90439,-123637,22599,88102,26907
C00829=-80407,-121901,-119741,18448,66455,46046
C00830=-99207,-113247,-119914,5586,82670,39005
C00831=-101996,-106609,-115785,6360,83734,38140
C00832=-119008,-118478,-113260,32340,76336,33375
C00833=-80488,-121328,-114439,18908,63658,45548
C00834=-79672,-120202,-114057,18494,63797,45891
C00835=-79592,-120276,-114079,18461,63755,45915
C00836=-80475,-121542,-115946,18779,64427,45684
C00837=-80482,-121578,-119613,18469,66554,46034
C00838=-85156,-144709,-129107,-21632,59402,64028
C00839=-93856,-120445,-109825,-39450,57641,70752
C00840=-93847,-119691,-106928,-40019,56559,71233
C00841=-86628,-99816,-98593,-45940,69277,74290
C00842=-86043,-99167,-98859,-45014,69635,74495
C00843=-83318,-93529,-94650,-47165,68336,75996
C00844=-93680,-116508,-100417,-40719,46210,72415
C00845=-93820,-118277,-102341,-40471,46353,72255
C00846=-93828,-119232,-105178,-39715,47322,71755
C00847=-93822,-120125,-107980,-28359,52237,38282
C00848=-93816,-119582,-106091,-28689,51458,38525
C00849=-93813,-119346,-105328,-28822,51152,38622
C00850=-93805,-118409,-102529,-29499,49391,39302
C00851=-93820,-119862,-107056,-29266,59584,40856
C00852=-93823,-120114,-107958,-29147,59957,40747
C00853=-93830,-120670,-110185,-28854,60909,40473
C00854=-63807,-119595,-131717,-32346,77391,31957
C00855=-66677,-121755,-125547,-9668,69981,-32239
C00856=-66675,-122709,-116301,-10101,63887,-31721
C00857=-66675,-122586,-115330,-10147,63360,-31673
C00858=-66678,-122782,-121307,9429,81851,-37654
C00859=-66765,-122962,-121469,9451,81867,-37681
C00860=-66675,-122328,-113778,33290,107246,-42961
C00861=-66675,-122499,-114776,33395,107690,-42822
C00862=-66677,-122795,-117228,33681,108831,-42458
C00863=-67830,-119002,-127241,35733,116022,-40496
C00864=-66677,-118144,-130351,-9432,74728,-32617
C00865=-66675,-122709,-116301,-10101,63887,-31721
C00866=-66675,-122566,-115195,-10154,63288,-31666
C00867=-66598,-122626,-121075,9408,81779,-37632
C00868=-62201,-135334,-124977,8438,77219,-36455
C00869=-72037,-126014,-118725,27283,91958,-49043
C00870=-76379,-123759,-128626,28058,99823,-48794
C00871=-71006,-123079,-126009,31798,108132,-44322
C00872=-66720,-122114,-124411,34847,112827,-41144
C00873=-125074,-112778,-121368,18538,134713,-61704
C00874=-173715,-145384,-131232,-10200,126221,-84589
C00875=-173715,-147046,-136936,-18176,117071,-78230
C00876=-173715,-145384,-131232,-55285,56270,-43989
C00877=-121435,-145384,-131232,-55285,56270,-43989
C00878=-118035,-115309,-97908,-59229,55500,-40903
C00879=-125649,-158907,-99513,-82423,43353,-29623
C00880=-115891,-110152,-98721,-57727,100769,-36262
C00881=-114349,-140479,-107559,-55988,95957,-32016
C00882=-114314,-138547,-101727,-57982,106397,-39425
C00883=-102008,-144788,-123359,-59173,119414,-41279
C00884=-15972,-110889,-128286,-10965,59905,-43045
C00885=-15972,-110889,-128286,-10965,59905,-43045
C00886=-101389,-60822,-75148,6919,68546,-70102
C00887=-115790,69230,64798,-8053,66131,-71909
C00888=-120688,105020,73307,-12402,84846,-73777
C00889=-120868,103639,75593,-12409,82749,-73629
C00890=-120940,103216,76680,-12418,81872,-73566
C00891=-120940,103732,79019,-12450,80724,-73451
C00892=-120940,103216,76680,-12418,81872,-73566
C00893=-120298,112004,89967,-12640,78393,-72988
C00894=-120707,106255,82361,-12511,80017,-73298
C00895=-120298,112004,89967,-12640,78393,-72988
C00896=-120228,112105,88453,-12614,79365,-73063
C00897=-120053,112844,85327,-12571,81642,-73235
C00898=-120830,71540,61874,-4756,55589,-66514
C00899=-120535,76858,72419,-5134,51864,-66212
C00900=-120418,79487,77321,-5314,50212,-66075
C00901=-120418,81305,81326,-5435,48689,-65991
C00902=-120418,79487,77321,-5314,50212,-66075
C00903=-121101,73566,71896,-4942,50464,-66384
C00904=-120640,77942,77238,-5256,49458,-66131
C00905=-121101,73566,71896,-4942,50464,-66384
C00906=-121222,71175,67349,-4775,52021,-66512
C00907=-121527,66226,57370,-4418,55590,-66797
C00908=-120817,46858,51705,6808,46216,-80289
C00909=-120487,52530,62238,7041,42645,-80409
C00910=-120357,55197,66992,7170,41090,-80474
C00911=-120357,57219,71131,7393,39594,-80606
C00912=-120357,55197,66992,7170,41090,-80474
C00913=-121171,51687,64922,7778,40638,-80922
C00914=-120657,55397,69123,7546,39918,-80729
C00915=-121171,51687,64922,7778,40638,-80922
C00916=-121307,49062,60252,7635,42163,-80850
C00917=-121648,43436,49847,7373,45678,-80715
C00918=-109578,66950,51259,-9202,73878,-70224
C00919=-101389,-60822,-75148,6919,68546,-70102
C00920=-96929,-90691,-89138,5080,61517,-23019
C00921=-96929,-90691,-89138,5080,61517,27168
C00922=-133997,38575,-5386,4879,105902,64390
C00923=-134430,35731,-4221,4855,103756,64161
C00924=-134605,34666,-3678,4847,102887,64068
C00925=-134604,34193,-2477,4825,101908,64030
C00926=-134605,34666,-3678,4847,102887,64068
C00927=-133324,38381,1851,4717,101326,64430
C00928=-133984,36157,-436,4773,101627,64224
C00929=-133324,38381,1851,4717,101326,64430
C00930=-132740,42105,45,4739,104308,64739
C00931=-159526,23962,790,32225,80504,55500
C00932=-158922,24925,5721,32299,78113,55050
C00933=-158682,25453,8443,32390,76826,54772
C00934=-158681,25549,9587,32465,76269,54609
C00935=-158682,25408,7790,32348,77149,54866
C00936=-160104,22984,7189,32780,76948,54233
C00937=-159169,24509,8648,32575,76492,54477
C00938=-160104,22984,7189,32780,76948,54233
C00939=-160967,21427,101,32642,80299,54873
C00940=-147551,27169,-6215,28445,81493,60312
C00941=-147017,27605,-1759,28452,79091,59917
C00942=-146805,27803,661,28506,77793,59674
C00943=-146803,27699,1600,28565,77235,59535
C00944=-146805,27874,109,28472,78126,59757
C00945=-148390,24338,-1607,29025,77984,59121
C00946=-147556,26192,183,28786,77573,59333
C00947=-148390,24338,-1607,29025,77984,59121
C00948=-149162,23542,-7999,28991,81344,59682
C00949=-129846,-17397,-52274,16165,101048,68229
C00950=-103949,-6271,-30701,7884,96105,76175
C00951=-94102,16895,-5866,4380,94047,79161
C00952=-94024,14878,-3719,4358,91692,79105
C00953=-93993,14152,-2780,4351,90742,79083
C00954=-93993,14253,-1030,4349,89719,79047
C00955=-93993,14152,-2780,4351,90742,79083
C00956=-93685,20015,4382,4321,89334,79138
C00957=-93881,17120,1686,4338,89515,79078
C00958=-93685,20015,4382,4321,89334,79138
C00959=-93796,22544,1176,4343,92603,79213
C00960=-95224,-25687,-42365,27028,60157,72238
C00961=-94111,-23276,-36997,26973,57954,72128
C00962=-93676,-22245,-34794,26967,57075,72081
C00963=-93677,-22196,-33100,27266,56165,71832
C00964=-93676,-22245,-34794,26967,57075,72081
C00965=-94165,-26445,-35973,27662,55954,71554
C00966=-93910,-23559,-33944,27450,56079,71704
C00967=-94165,-26445,-35973,27662,55954,71554
C00968=-95768,-30118,-43626,27714,58991,71694
C00969=-97625,-41604,-59467,17173,89706,-8843
C00970=-96114,-37688,-53918,16886,88057,-8555
C00971=-95526,-36022,-51615,16777,87400,-8443
C00972=-95527,-36150,-50037,16784,86406,-8579
C00973=-95526,-36022,-51615,16777,87400,-8443
C00974=-95532,-36183,-50637,16782,86745,-8534
C00975=-95234,-33170,-48668,16723,87008,-8396
C00976=-95532,-36183,-50637,16782,86745,-8534
C00977=-95504,-36095,-50208,16778,86530,-8554
C00978=-93996,-36675,-50581,16493,86163,-8084
C00979=-95504,-36095,-50208,16778,86530,-8554
C00980=-97625,-41604,-59467,17173,89706,-8843
C00981=-101873,-77751,-87156,42969,63075,62474
C00982=-95937,-74809,-81328,40948,58735,63434
C00983=-95565,-74583,-80935,40815,58468,63500
C00984=-95566,-74620,-79294,41227,57681,63141
C00985=-95565,-74583,-80935,40815,58468,63500
C00986=-98755,-73227,-80296,42221,60183,62682
C00987=-98803,-73638,-78797,42678,59356,62269
C00988=-96868,-74481,-79195,41849,58298,62761
C00989=-98803,-73638,-78797,42678,59356,62269
C00990=-97163,-69666,-76891,41573,59236,63045
C00991=-96752,-66139,-75134,41097,59602,63417
C00992=-97163,-69666,-76891,41573,59236,63045
C00993=-101873,-77751,-87156,42969,63075,62474
C00994=-126113,-49786,-51573,51544,90004,55144
C00995=-123973,-50127,-48217,51392,87374,54806
C00996=-123286,-49758,-46380,51349,86473,54664
C00997=-118478,-34750,-37348,50925,85086,56432
C00998=-119272,-35479,-39244,50973,86038,56539
C00999=-121232,-35158,-42579,51146,88553,56901
C01000=-111145,-57425,-62081,41633,61582,55088
C01001=-109620,-53993,-56645,41578,59663,54986
C01002=-109014,-52418,-54338,41560,58914,54950
C01003=-105531,-54881,-55720,40219,56972,55856
C01004=-106107,-56401,-57979,40230,57706,55889
C01005=-107578,-60042,-63488,40293,59558,55964
C01006=-93331,-25535,-46307,22677,87971,72102
C01007=-84242,-5399,-27465,11713,100257,81196
C01008=-83743,-8192,-25851,11599,97806,81134
C01009=-83603,-8644,-24372,11558,96668,81075
C01010=-80847,-8673,-24279,11462,96208,81977
C01011=-80973,-8366,-25985,11504,97411,82047
C01012=-81511,-5615,-27635,11617,99868,82095
C01013=-103949,-6271,-30701,7884,96105,76175
C01014=-129846,-17397,-52274,16165,101048,68229
C01015=-175693,57260,35469,48998,74273,48315
C01016=-174652,59964,42108,49342,71909,47593
C01017=-173987,58917,42535,48748,68669,47097
C01018=-173562,58305,42809,47399,62634,46211
C01019=-173482,53917,36869,46602,62532,46609
C01020=-174364,49990,29079,45939,64941,47387
C01021=-163099,39792,11105,47007,80916,54866
C01022=-161954,40669,15666,46993,78691,54338
C01023=-161675,41954,18470,47071,77805,54042
C01024=-160520,35916,12218,46685,77730,54566
C01025=-160850,34862,9687,46632,78611,54832
C01026=-162019,34035,5199,46665,80839,55343
C01027=-147988,42797,109,12455,106225,61454
C01028=-148219,40121,1423,12320,104123,61157
C01029=-148209,38525,1410,12269,103328,61081
C01030=-147238,35306,-1899,12234,103563,61431
C01031=-146513,33084,-4151,12206,103702,61693
C01032=-146794,35355,-3496,12271,104485,61677
C01033=-146567,38090,-4821,12411,106625,61976
C01034=-96929,-90691,-89138,5080,61517,27168
C01035=-96929,-90691,-89138,5080,61517,-23019
C01036=-101389,-60822,-75148,6919,68546,-70102
C01037=-109578,66950,51259,-9202,73878,-70224
C01038=-119285,73548,61078,-7759,54489,-67872
C01039=-119140,78931,71700,-8230,50768,-67516
C01040=-119083,81584,76629,-8462,49121,-67350
C01041=-122917,98444,98202,-6801,44189,-68705
C01042=-122308,90513,86215,-6785,47517,-68668
C01043=-122473,83260,72935,-6271,51921,-69036
C01044=-119074,82203,59752,-14757,75142,-72556
C01045=-112473,77653,55392,-16315,76732,-70397
C01046=-111583,66581,50085,-22599,68947,-68307
C01047=-112205,67748,51306,-22435,68636,-68485
C01048=-112291,70891,55012,-22505,67993,-68392
C01049=-120890,75924,58725,-8799,66214,-71114
C01050=-120891,72538,54662,-8752,66965,-71172
C01051=-121396,73617,55948,-8591,66676,-71337
C01052=-121396,72779,51526,-8459,68942,-71502
C01053=-134157,70152,49704,15847,72235,-43808
C01054=-133722,73949,59265,16087,68355,-44178
C01055=-133862,75249,62165,16247,67307,-44381
C01056=-129675,65866,51066,4701,64817,-31992
C01057=-128682,62362,47014,4314,65455,-31601
C01058=-130205,57581,36634,4742,69462,-32000
C01059=-130312,54578,33992,4779,69550,-32035
C01060=-129992,46081,35923,20239,67004,8502
C01061=-121496,43425,36833,5893,59088,22773
C01062=-120237,47252,43120,2387,56768,25932
C01063=-119972,47626,45454,2298,55515,26011
C01064=-128073,50557,47782,20949,62737,7811
C01065=-127834,53853,52717,21124,61417,7650
C01066=-123180,48310,46556,9691,56439,19302
C01067=-122651,35401,27095,8965,61652,19959
C01068=-109578,66950,51259,-9202,73878,-70224
C01069=-101389,-60822,-75148,6919,68546,-70102
C01070=-96929,-90691,-89138,5080,61517,-23019
C01071=-93242,-109726,-96296,3420,55961,28393
C01072=-92156,-22649,-39625,10516,94476,60392
C01073=-92549,-23820,-36378,10508,91967,60047
C01074=-92689,-24290,-35079,10509,90961,59915
C01075=-95254,-23373,-34430,10727,91365,59075
C01076=-94898,-22950,-35761,10710,92338,59280
C01077=-94492,-21797,-39017,10723,94837,59633
C01078=-92575,-26977,-42679,21088,73618,56030
C01079=-92430,-25186,-37423,21282,71416,55682
C01080=-92290,-24713,-35488,21345,70493,55566
C01081=-95616,-23226,-34216,23502,71566,54461
C01082=-95477,-23933,-36320,23344,72386,54682
C01083=-95719,-25683,-41558,23174,74597,55037
C01084=-96929,-90691,-89138,5080,61517,27168
C01085=-96929,-90691,-89138,5080,61517,-23019
C01086=-101389,-60822,-75148,6919,68546,-70102
C01087=-109578,66950,51259,-9202,73878,-70224
C01088=-108278,48890,46404,-6655,48460,-73563
C01089=-108252,54023,56228,-7048,45078,-73302
C01090=-108672,56895,61153,-6970,43500,-73378
C01091=-113114,65075,70630,-4174,41573,-75428
C01092=-112702,61866,65174,-4315,43297,-75310
C01093=-112766,56024,54314,-4011,46966,-75508
C01094=-103921,32533,46603,10708,30188,-75698
C01095=-104692,35200,60863,30413,16065,-83251
C01096=-104796,38679,66061,33302,14894,-84599
C01097=-102333,36267,63497,27606,14351,-81669
C01098=-100412,37194,55383,7603,26828,-73795
C01099=-100998,29868,43914,7479,30147,-73786
C01100=-109578,66950,51259,-9202,73878,-70224
C01101=-101389,-60822,-75148,6919,68546,-70102
C01102=-96929,-90691,-89138,5080,61517,-23019
C01103=-96929,-90691,-89138,5080,61517,27168
C01104=-90570,-23240,-39845,-1682,91658,61068
C01105=-90349,-1837,-19216,-4288,101242,62233
C01106=-90005,-3734,-19299,-4261,100340,62382
C01107=-92752,-2865,-18588,-4343,100202,61442
C01108=-95291,-22836,-35623,-1093,89189,59526
C01109=-94239,-22001,-38963,-1226,91687,59852
C01110=-90424,-29050,-43505,3763,58999,61302
C01111=-86008,-21130,-36360,-6353,62529,61992
C01112=-86454,-19207,-33152,-6175,61515,61881
C01113=-89453,-18520,-32647,-4592,61359,60761
C01114=-95351,-24457,-36663,6763,57473,59317
C01115=-94707,-27619,-42528,6252,59394,59681
C01116=-109011,-26713,-50438,8452,98222,74634
C01117=-144543,31549,-11380,-159,92982,60584
C01118=-143093,45679,4448,-4866,97184,60249
C01119=-143214,43522,5393,-4827,95492,60276
C01120=-146471,54490,17318,-4285,93619,59288
C01121=-148937,42537,3991,922,89189,59187
C01122=-148250,43318,770,754,91565,59420
C01123=-172279,3947,-14828,46151,77384,48319
C01124=-167570,-10636,-17777,41693,62852,42800
C01125=-166655,-7092,-11488,42082,60867,42363
C01126=-169056,5005,-1455,42887,62060,41693
C01127=-172859,17944,7820,47479,72977,45875
C01128=-174013,15583,1984,47261,75226,46421
C01129=-109011,-26713,-50438,8452,98222,74634
C01130=-99312,-50897,-61026,22837,72179,74454
C01131=-98138,-49989,-56545,22703,69739,74412
C01132=-106382,-52347,-50887,37007,65807,70627
C01133=-98813,-18962,-39289,22939,92751,75811
C01134=-101547,-27333,-44313,25543,91651,74875
C01135=-97857,-18198,-39852,20610,99055,76884
C01136=-96922,-25876,-47272,18742,95048,76352
C01137=-97638,-23312,-49453,18962,97729,76524
C01138=-81141,-50558,-66105,12803,46081,75388
C01139=-80687,-46119,-60183,12697,44679,75401
C01140=-80513,-44339,-57785,12667,44105,75401
C01141=-80516,-44488,-54802,13120,42239,75121
C01142=-80690,-46329,-57233,13145,42803,75122
C01143=-81145,-50923,-63237,13239,44177,75109
C01144=-83601,15534,-39616,9664,96262,77072
C01145=-80484,90945,50155,4324,118905,78550
C01146=-80490,84570,45509,4303,118490,78531
C01147=-80493,82108,43801,4293,118276,78521
C01148=-80495,81630,46278,4216,116511,78452
C01149=-80492,84058,47940,4226,116735,78462
C01150=-83493,53381,-2692,9637,111099,78940
C01151=-91945,-14209,-43630,9790,83010,75128
C01152=-10907,-117335,-90652,-18762,63715,-59495
C01153=-15972,-110889,-128286,-10965,59905,-43045
BC00000=48829,688840,1075175
BC00001=366911,902233,1075175
BC00002=366911,902233,1075175
BC00003=366911,902233,1075175
BC00004=366911,902233,1075175
BC00005=366911,902233,1075175
BC00006=366911,902233,1075175
BC00007=366911,902233,1075175
BC00008=366911,902233,1075175
BC00009=333056,895412,1075175
BC00010=333056,895412,1075175
BC00011=333056,895412,1075175
BC00012=333056,895412,1075175
BC00013=333056,895412,1075175
BC00014=333056,895412,1075175
BC00015=333056,895412,1075175
BC00016=333056,895412,1075175
BC00017=358091,902222,1075175
BC00018=358091,902222,1075175
BC00019=358091,902222,1075175
BC00020=358091,902222,1075175
BC00021=358091,902222,1075175
BC00022=358091,902222,1075175
BC00023=358091,902222,1075175
BC00024=358091,902222,1075175
BC00025=358091,902222,1075175
BC00026=358091,902222,1075175
BC00027=358091,902222,1075175
BC00028=358091,902222,1075175
BC00029=358091,902222,1075175
BC00030=358091,902222,1075175
BC00031=398174,894103,1075175
BC00032=398174,894103,1075175
BC00033=398174,894103,1075175
BC00034=398174,894103,1075175
BC00035=398174,894103,1075175
BC00036=398174,894103,1075175
BC00037=398174,894103,1075175
BC00038=398174,894103,1075175
BC00039=264903,781270,1075175
BC00040=264903,781270,1075175
BC00041=264904,781269,1075172
BC00042=264904,781269,1075171
BC00043=264904,781269,1075171
BC00044=264904,781269,1075168
BC00045=264904,781269,1075168
BC00046=264904,781269,1075168
BC00047=264904,781269,1075168
BC00048=264904,781269,1075168
BC00049=264904,781269,1075164
BC00050=264903,781270,1075175
BC00051=301264,775814,1075175
BC00052=301264,775814,1075175
BC00053=301264,775814,1075175
BC00054=301264,775814,1075175
BC00055=301264,775814,1075175
BC00056=301264,775814,1075175
BC00057=301264,775814,1075175
BC00058=301264,775814,1075175
BC00059=301264,775814,1075175
BC00060=301264,775814,1075175
BC00061=274235,786209,1075175
BC00062=238672,799885,1075175
BC00063=238672,799885,1075175
BC00064=238672,799885,1075175
BC00065=238672,799885,1075175
BC00066=238672,799885,1075175
BC00067=238672,799885,1075175
BC00068=238672,799885,1075175
BC00069=238672,799885,1075175
BC00070=238672,799884,1075171
BC00071=238672,799884,1075171
BC00072=238672,799885,1075175
BC00073=238672,799885,1075175
BC00074=238672,799885,1075175
BC00075=238672,799885,1075175
BC00076=318263,750454,1075175
BC00077=318263,750454,1075175
BC00078=318263,750454,1075175
BC00079=318263,750454,1075175
BC00080=318263,750454,1075175
BC00081=318263,750454,1075175
BC00082=318263,750454,1075175
BC00083=318263,750454,1075175
BC00084=318263,750454,1075175
BC00085=318263,750454,1075175
BC00086=318263,750454,1075175
BC00087=318263,750454,1075175
BC00088=318263,750454,1075175
BC00089=318263,750454,1075175
BC00090=318263,750454,1075175
BC00091=318263,750454,1075175
BC00092=318263,750454,1075175
BC00093=318263,750454,1075175
BC00094=318263,750454,1075175
BC00095=318263,750454,1075175
BC00096=318263,750454,1075175
BC00097=318263,750454,1075175
BC00098=318263,750454,1075175
BC00099=318263,750454,1075175
BC00100=318263,750454,1075175
BC00101=377114,750454,1075175
BC00102=397814,750454,1075175
BC00103=397814,750454,1075175
BC00104=397814,750454,1075175
BC00105=397814,750454,1075175
BC00106=397814,750454,1075175
BC00107=397814,750454,1075175
BC00108=397814,750454,1075175
BC00109=397814,750454,1075175
BC00110=397814,750454,1075175
BC00111=397814,750454,1075175
BC00112=397814,750454,1075175
BC00113=397814,750454,1075175
BC00114=397814,750454,1075175
BC00115=397814,750454,1075175
BC00116=397814,750454,1075175
BC00117=397814,750454,1075175
BC00118=397814,750454,1075175
BC00119=397814,750454,1075175
BC00120=397814,750454,1075175
BC00121=397814,750454,1075175
BC00122=383090,762961,1075175
BC00123=372387,772052,1075175
BC00124=296274,836703,1075175
BC00125=296274,836703,1075175
BC00126=296274,836703,1075175
BC00127=296274,836703,1075175
BC00128=296274,836703,1075175
BC00129=296274,836703,1075175
BC00130=296274,836703,1075175
BC00131=296274,836703,1075175
BC00132=296274,836703,1075175
BC00133=296274,836703,1075175
BC00134=296274,836703,1075175
BC00135=296274,836703,1075175
BC00136=296274,836703,1075175
BC00137=312215,899988,1075175
BC00138=312215,944285,1075175
BC00139=312215,944285,1075175
BC00140=312215,944285,1075175
BC00141=312215,944285,1075175
BC00142=312215,944285,1075175
BC00143=312215,944285,1075175
BC00144=312215,944285,1075175
BC00145=312215,944285,1075175
BC00146=312215,944285,1075175
BC00147=312215,944285,1075175
BC00148=312215,944285,1075175
BC00149=312215,944285,1075175
BC00150=312215,944285,1075175
BC00151=312215,944285,1075175
BC00152=312215,944285,1075175
BC00153=312215,944285,1075175
BC00154=312215,944285,1075175
BC00155=312215,944285,1075175
BC00156=287266,941775,1075175
BC00157=287266,941775,1075175
BC00158=287266,941775,1075175
BC00159=287266,941775,1075175
BC00160=287266,941775,1075175
BC00161=287266,941775,1075175
BC00162=259299,938961,1075175
BC00163=259299,938961,1075175
BC00164=259299,938961,1075175
BC00165=259299,938961,1075175
BC00166=259299,938961,1075175
BC00167=259299,938961,1075175
BC00168=259299,938961,1075175
BC00169=259299,938961,1075175
BC00170=259299,938961,1075175
BC00171=259299,938961,1075175
BC00172=259299,938961,1075175
BC00173=259299,938961,1075175
BC00174=211531,951911,1075175
BC00175=211531,951911,1075175
BC00176=211531,951911,1075175
BC00177=211531,951911,1075175
BC00178=211531,951911,1075175
BC00179=211531,951911,1075175
BC00180=211531,951913,1075174
BC00181=314656,958350,1075174
BC00182=314656,958350,1075174
BC00183=314656,958350,1075174
BC00184=314656,958350,1075174
BC00185=314656,958350,1075174
BC00186=314656,958350,1075174
BC00187=314656,958350,1075174
BC00188=314656,958350,1075174
BC00189=314656,958350,1075174
BC00190=314656,958350,1075174
BC00191=314656,958350,1075174
BC00192=211531,951911,1075175
BC00193=211531,951911,1075175
BC00194=211531,951911,1075175
BC00195=211531,951911,1075175
BC00196=211531,951911,1075175
BC00197=211531,951911,1075175
BC00198=211531,951911,1075175
BC00199=211531,951912,1075174
BC00200=211531,951912,1075174
BC00201=211531,951912,1075174
BC00202=211531,951912,1075174
BC00203=211531,951912,1075174
BC00204=211531,951912,1075174
BC00205=211531,951912,1075174
BC00206=211531,951912,1075174
BC00207=211531,951912,1075174
BC00208=211531,951912,1075174
BC00209=182503,951872,1075175
BC00210=184369,953383,1075175
BC00211=184369,953399,1075175
BC00212=184333,953526,1075175
BC00213=184897,956550,1075175
BC00214=184333,953526,1075175
BC00215=184751,953664,1075175
BC00216=187887,953121,1075175
BC00217=184751,953664,1075175
BC00218=178222,948378,1075175
BC00219=171711,951911,1075175
BC00220=174897,958670,1075175
BC00221=174897,958670,1075175
BC00222=174897,958670,1075175
BC00223=174897,958670,1075175
BC00224=174897,958672,1075174
BC00225=278022,965109,1075174
BC00226=278022,965109,1075174
BC00227=278022,965109,1075174
BC00228=278022,965109,1075174
BC00229=278022,965109,1075174
BC00230=278022,965109,1075174
BC00231=278022,965109,1075174
BC00232=278022,965109,1075174
BC00233=278022,965109,1075174
BC00234=278022,965109,1075174
BC00235=278022,965109,1075174
BC00236=174897,958670,1075175
BC00237=174897,958670,1075175
BC00238=174897,958670,1075175
BC00239=174897,958670,1075175
BC00240=174897,958670,1075175
BC00241=174897,958670,1075175
BC00242=174897,958670,1075175
BC00243=174897,958671,1075174
BC00244=174897,958671,1075174
BC00245=174897,958671,1075174
BC00246=174897,958671,1075174
BC00247=174897,958671,1075174
BC00248=174897,958671,1075174
BC00249=174897,958671,1075174
BC00250=174897,958671,1075174
BC00251=174897,958671,1075174
BC00252=174897,958671,1075174
BC00253=182815,952263,1075175
BC00254=183711,957103,1075175
BC00255=184069,959047,1075174
BC00256=184070,959056,1075175
BC00257=184189,959079,1075175
BC00258=184752,962103,1075175
BC00259=184189,959079,1075175
BC00260=182935,952303,1075175
BC00261=182935,952303,1075175
BC00262=182935,952303,1075175
BC00263=123088,1061215,1075175
BC00264=126332,1055781,1075175
BC00265=127630,1053613,1075175
BC00266=127630,1053623,1075175
BC00267=127630,1053607,1075175
BC00268=153753,1064749,1075175
BC00269=152152,1062093,1075175
BC00270=153753,1064749,1075175
BC00271=104366,1038154,1075175
BC00272=107120,1036610,1075175
BC00273=104366,1038154,1075175
BC00274=97490,1044180,1075175
BC00275=121157,1044973,1075175
BC00276=140343,1045718,1075175
BC00277=158643,1046375,1075175
BC00278=155464,1041036,1075175
BC00279=155106,1040455,1075175
BC00280=155106,1040463,1075175
BC00281=155288,1040367,1075175
BC00282=153687,1037711,1075175
BC00283=155288,1040367,1075175
BC00284=158891,1046297,1075175
BC00285=211337,993614,1075175
BC00286=274623,983932,1075175
BC00287=371761,1043051,1075175
BC00288=331941,1063020,1075175
BC00289=331941,1063020,1075175
BC00290=331941,1063020,1075175
BC00291=331941,1063020,1075175
BC00292=331941,1063020,1075175
BC00293=331941,1063020,1075175
BC00294=331941,1063020,1075175
BC00295=331941,1063020,1075175
BC00296=331941,1063020,1075175
BC00297=331941,1063020,1075175
BC00298=331941,1063020,1075175
BC00299=331941,1063020,1075175
BC00300=344464,1061929,1051932
BC00301=344464,1061928,1051932
BC00302=344464,1061928,1051932
BC00303=344464,1061928,1051932
BC00304=344464,1061928,1051932
BC00305=344464,1061928,1051932
BC00306=344464,1061928,1051932
BC00307=344464,1061928,1051932
BC00308=328139,1011393,1051932
BC00309=328139,1011393,1051932
BC00310=328139,1011393,1051932
BC00311=328139,1011393,1051932
BC00312=328139,1011393,1051932
BC00313=328139,1011393,1051932
BC00314=328139,1011393,1051932
BC00315=328139,1011393,1051932
BC00316=331941,1063020,1075175
BC00317=331941,1063020,1075175
BC00318=371761,1043051,1075175
BC00319=371761,1043051,1075175
BC00320=371761,1043051,1075175
BC00321=371761,1043051,1075175
BC00322=371761,1043051,1075175
BC00323=371761,1043051,1075175
BC00324=371761,1043051,1075175
BC00325=371761,1043051,1075175
BC00326=371761,1043051,1075175
BC00327=371761,1043051,1075175
BC00328=371761,1043051,1075175
BC00329=371761,1043051,1075175
BC00330=371761,1043051,1075175
BC00331=371761,1043051,1075175
BC00332=371761,1043051,1075175
BC00333=314185,938855,1075175
BC00334=247671,970611,1075175
BC00335=247671,970611,1075175
BC00336=247671,970611,1075175
BC00337=247671,970611,1075175
BC00338=247671,970611,1075175
BC00339=247671,970611,1075175
BC00340=247671,970611,1075175
BC00341=247671,970611,1075175
BC00342=247671,970611,1075175
BC00343=247671,970611,1075175
BC00344=247671,970611,1075175
BC00345=247671,970611,1075175
BC00346=207145,985111,1075175
BC00347=158336,1040306,1075175
BC00348=208463,1020843,1075175
BC00349=208463,1020843,1075175
BC00350=208462,1020843,1075174
BC00351=208462,1020843,1075174
BC00352=208462,1020843,1075174
BC00353=208462,1020843,1075174
BC00354=229380,1020843,1075174
BC00355=229380,1020843,1075174
BC00356=229380,1020843,1075174
BC00357=229380,1020843,1075174
BC00358=229380,1020843,1075174
BC00359=229380,1020843,1075174
BC00360=303037,872055,1075175
BC00361=380992,820655,1075175
BC00362=380992,820655,1075175
BC00363=380992,820655,1075175
BC00364=380992,820655,1075175
BC00365=380992,820655,1075175
BC00366=380992,820655,1075175
BC00367=380992,820655,1075175
BC00368=380992,820655,1075175
BC00369=380992,820655,1075175
BC00370=380992,820655,1075175
BC00371=380992,820655,1075175
BC00372=380992,820655,1075175
BC00373=275256,812324,1075175
BC00374=275256,839586,1075175
BC00375=275256,839586,1074242
BC00376=275256,839586,1074242
BC00377=275256,839586,1074242
BC00378=275256,839586,1074242
BC00379=275256,812324,1075175
BC00380=125716,897903,1075175
BC00381=125716,897903,1075175
BC00382=125716,897903,1075175
BC00383=125716,897903,1075175
BC00384=125716,897903,1075175
BC00385=125716,897903,1075174
BC00386=125716,897903,1075171
BC00387=125716,897903,1075175
BC00388=125716,897903,1075175
BC00389=125716,897903,1075175
BC00390=125716,897903,1075175
BC00391=125716,897903,1075175
BC00392=125716,897903,1075175
BC00393=325019,822543,1075229
BC00394=325019,822543,1075229
BC00395=325019,822543,1075229
BC00396=325019,822543,1075229
BC00397=325019,822543,1075229
BC00398=325019,822543,1075229
BC00399=325019,822543,1075229
BC00400=325019,822543,1075229
BC00401=325019,822543,1075229
BC00402=325019,822543,1075229
BC00403=325019,822543,1075229
BC00404=325019,822543,1075229
BC00405=240667,871930,1075210
BC00406=81335,965219,1075175
BC00407=81335,965219,1075175
BC00408=81335,965219,1075175
BC00409=81335,965219,1075175
BC00410=81335,965219,1075175
BC00411=81335,965219,1075175
BC00412=81335,965219,1075175
BC00413=81335,965219,1075175
BC00414=39891,972466,1075175
BC00415=39891,972466,1075175
BC00416=39891,972466,1075175
BC00417=39891,972466,1075175
BC00418=39891,972466,1075175
BC00419=39891,972466,1075175
BC00420=39891,972466,1075175
BC00421=39891,1005107,1075175
BC00422=39891,1005107,1075175
BC00423=39891,1005107,1075175
BC00424=39891,1005107,1075175
BC00425=39891,1005107,1075175
BC00426=39891,1005107,1075175
BC00427=39891,972466,1075175
BC00428=126064,942124,1075175
BC00429=145718,951183,1075175
BC00430=145718,951183,1075175
BC00431=145718,951183,1075175
BC00432=145718,951183,1075175
BC00433=145718,951183,1075175
BC00434=145718,951183,1075175
BC00435=145718,951183,1075175
BC00436=145718,951183,1075175
BC00437=145718,951183,1075175
BC00438=145718,951183,1075175
BC00439=145718,951183,1075175
BC00440=145718,951183,1075175
BC00441=127193,914007,1075175
BC00442=75497,867475,1075175
BC00443=75497,867475,1075175
BC00444=75497,867475,1075175
BC00445=75497,867475,1075175
BC00446=75497,867475,1075175
BC00447=75497,867475,1075175
BC00448=75497,867475,1075175
BC00449=75497,867475,1075175
BC00450=75497,867475,1075175
BC00451=75497,867475,1075175
BC00452=75497,867475,1075175
BC00453=75497,867475,1075175
BC00454=75497,867475,1075175
BC00455=75497,867475,1075175
BC00456=75497,867475,1075175
BC00457=75497,867475,1075175
BC00458=75497,867475,1075175
BC00459=58830,852413,1075175
BC00460=43274,838354,1075175
BC00461=43274,838354,1075175
BC00462=43274,838354,1075175
BC00463=43274,838354,1075175
BC00464=43274,838354,1075175
BC00465=43274,838354,1075175
BC00466=43274,838354,1075175
BC00467=43274,838354,1075175
BC00468=43274,838354,1075175
BC00469=191439,896290,1075175
BC00470=209593,874493,1075175
BC00471=209593,874493,1075175
BC00472=209593,874493,1075174
BC00473=209593,874493,1075171
BC00474=209593,874493,1075175
BC00475=209593,874493,1075175
BC00476=209216,850926,1075175
BC00477=226866,854473,1075175
BC00478=228835,855864,1075175
BC00479=228835,855864,1075175
BC00480=228834,855864,1075173
BC00481=228834,855864,1075173
BC00482=228835,855864,1075175
BC00483=228835,855864,1075175
BC00484=228835,855864,1075175
BC00485=228835,855864,1075175
BC00486=228835,855864,1075175
BC00487=212683,986357,1075175
BC00488=212683,1004517,1075175
BC00489=212247,999872,1075175
BC00490=212146,998778,1075171
BC00491=214955,996593,1075174
BC00492=222186,994128,1075175
BC00493=222622,998773,1075175
BC00494=293477,973063,1075175
BC00495=293477,973063,1075175
BC00496=293477,973063,1075175
BC00497=293477,973063,1075175
BC00498=293477,973063,1075175
BC00499=293477,973063,1075175
BC00500=293477,973063,1075175
BC00501=293477,973063,1075175
BC00502=248777,974412,1075175
BC00503=147624,1017934,1075175
BC00504=124950,1033375,1075175
BC00505=124950,1033375,1075175
BC00506=124950,1033375,1075175
BC00507=124950,1033375,1075174
BC00508=124950,1033375,1075175
BC00509=124950,1033375,1075175
BC00510=106678,1046165,1075175
BC00511=106678,1046165,1075175
BC00512=106678,1046165,1075175
BC00513=106678,1046165,1075175
BC00514=106678,1046165,1075175
BC00515=106678,1046165,1075175
BC00516=172863,1024486,1075175
BC00517=172427,1019841,1075175
BC00518=172326,1018747,1075171
BC00519=175135,1016562,1075174
BC00520=182366,1014097,1075175
BC00521=182802,1018742,1075175
BC00522=253657,993032,1075175
BC00523=253657,993032,1075175
BC00524=253657,993032,1075175
BC00525=253657,993032,1075175
BC00526=253657,993032,1075175
BC00527=253657,993032,1075175
BC00528=253657,993032,1075175
BC00529=253657,993032,1075175
BC00530=208957,994381,1075175
BC00531=107804,1037903,1075175
BC00532=85130,1053344,1075175
BC00533=85130,1053344,1075175
BC00534=85130,1053344,1075175
BC00535=85130,1053344,1075175
BC00536=85130,1053344,1075175
BC00537=85130,1053344,1075175
BC00538=66858,1066134,1075175
BC00539=66858,1066134,1075175
BC00540=66858,1066134,1075175
BC00541=66858,1066134,1075175
BC00542=66858,1066134,1075175
BC00543=66858,1066134,1075175
BC00544=106678,1034404,1075175
BC00545=288363,951317,1075175
BC00546=319880,932288,1075175
BC00547=316203,930177,1075175
BC00548=314732,929332,1075175
BC00549=314732,929332,1075175
BC00550=314732,929332,1075175
BC00551=294141,940882,1075174
BC00552=285351,949486,1075175
BC00553=280844,953897,1075175
BC00554=266486,999402,1075171
BC00555=253996,970793,1075175
BC00556=256777,973747,1075175
BC00557=224914,994659,1075175
BC00558=193407,1014756,1075175
BC00559=196552,1009267,1075175
BC00560=197065,1008372,1075175
BC00561=197397,1007797,1075175
BC00562=196552,1009278,1075175
BC00563=193407,1014766,1075175
BC00564=170876,1031134,1075175
BC00565=153007,1044116,1075175
BC00566=153007,1044116,1075175
BC00567=155599,1038213,1075175
BC00568=156636,1035851,1075175
BC00569=230598,1025728,1075175
BC00570=222023,1030515,1075175
BC00571=222023,1030515,1075175
BC00572=118655,1062836,1075175
BC00573=118655,1062836,1075175
BC00574=118655,1062836,1075175
BC00575=176896,1055708,1075175
BC00576=225377,1010635,1075175
BC00577=228184,1010601,1075175
BC00578=235201,1010515,1075175
BC00579=242597,980334,1075175
BC00580=282680,816770,1075175
BC00581=287393,774165,1075175
BC00582=293866,776192,1075175
BC00583=296455,777002,1075175
BC00584=296337,777088,1075175
BC00585=296308,777110,1075175
BC00586=296189,777197,1075175
BC00587=293600,776386,1075175
BC00588=287127,774359,1075175
BC00589=265173,805126,1075175
BC00590=271841,806848,1075175
BC00591=274508,807537,1075175
BC00592=274508,807537,1075175
BC00593=271842,806893,1075175
BC00594=265174,805171,1075175
BC00595=347775,809657,1075175
BC00596=348436,809459,1075175
BC00597=348700,809380,1075175
BC00598=352833,807067,1075175
BC00599=364813,800347,1075175
BC00600=368942,798027,1075175
BC00601=368677,798106,1075175
BC00602=368016,798304,1075175
BC00603=368016,798304,1075175
BC00604=391344,687000,1075175
BC00605=391344,687000,1075175
BC00606=391344,687000,1075175
BC00607=391344,687000,1075175
BC00608=391344,687000,1075175
BC00609=391344,687000,1075175
BC00610=391344,687000,1075175
BC00611=391344,687000,1075175
BC00612=391344,687000,1075175
BC00613=391344,687000,1075175
BC00614=391344,687000,1075175
BC00615=391344,687000,1075175
BC00616=358873,687000,1075175
BC00617=250171,896024,1075175
BC00618=255370,893912,1075175
BC00619=257449,893067,1075174
BC00620=259851,897051,1075175
BC00621=270502,914711,1075175
BC00622=268422,915555,1075175
BC00623=263223,917668,1075175
BC00624=251695,824506,1075175
BC00625=253916,829548,1075175
BC00626=254804,831565,1075175
BC00627=231448,844598,1075175
BC00628=231448,844598,1075175
BC00629=197017,859048,1075175
BC00630=197017,859048,1075175
BC00631=188570,860127,1075175
BC00632=185301,855336,1075175
BC00633=261332,833542,1075175
BC00634=297112,823286,1075175
BC00635=293523,829343,1075175
BC00636=292087,831765,1075175
BC00637=292088,831788,1075175
BC00638=293523,829365,1075175
BC00639=297112,823308,1075175
BC00640=297112,823286,1075175
BC00641=112345,954746,1075175
BC00642=112345,954746,1075175
BC00643=111546,959512,1075175
BC00644=111226,961418,1075175
BC00645=111226,961418,1075175
BC00646=111226,961418,1075175
BC00647=63698,969650,1075175
BC00648=63700,969637,1075175
BC00649=63700,969637,1075175
BC00650=63700,969637,1075175
BC00651=64817,962978,1075175
BC00652=55529,859309,1075175
BC00653=51595,858048,1075175
BC00654=50021,857544,1075175
BC00655=45895,833192,1075175
BC00656=46071,849801,1075175
BC00657=43912,844296,1075175
BC00658=45475,843733,1075175
BC00659=45475,843733,1075175
BC00660=45475,843733,1075175
BC00661=45475,843733,1075175
BC00662=45475,843733,1075175
BC00663=49382,842326,1075175
BC00664=32191,855540,1075175
BC00665=35199,856902,1075175
BC00666=36402,857447,1075175
BC00667=24170,872455,1075175
BC00668=24116,855865,1075175
BC00669=17601,856883,1075175
BC00670=10106,858388,1075175
BC00671=7107,859694,1075175
BC00672=124165,958731,1075175
BC00673=124477,964204,1075175
BC00674=124602,966393,1075175
BC00675=119899,967208,1075175
BC00676=119804,967224,1075175
BC00677=119804,967224,1075175
BC00678=114534,965927,1075175
BC00679=114222,960453,1075175
BC00680=169497,963360,1075175
BC00681=218455,965934,1075175
BC00682=214431,967961,1075175
BC00683=212822,968772,1075175
BC00684=212822,968772,1075175
BC00685=212822,968772,1075175
BC00686=218344,963319,1075175
BC00687=222368,961291,1075175
BC00688=147324,958268,1075175
BC00689=86350,984014,1075175
BC00690=90717,985390,1075175
BC00691=92241,985755,1075175
BC00692=87949,982178,1075175
BC00693=87949,982178,1075175
BC00694=86202,981627,1075175
BC00695=81835,980250,1075175
BC00696=83182,969192,1075175
BC00697=84657,971884,1075175
BC00698=84782,974073,1075175
BC00699=84782,974073,1075175
BC00700=84664,974093,1075175
BC00701=84664,974093,1075175
BC00702=74714,973607,1075175
BC00703=74402,968133,1075175
BC00704=129677,971040,1075175
BC00705=178635,973614,1075175
BC00706=174611,975641,1075175
BC00707=173002,976452,1075175
BC00708=173002,976452,1075175
BC00709=173002,976452,1075175
BC00710=178524,970999,1075175
BC00711=182548,968971,1075175
BC00712=107504,965948,1075175
BC00713=46530,991694,1075175
BC00714=50897,993070,1075175
BC00715=52421,993435,1075175
BC00716=52296,993331,1075175
BC00717=52254,993296,1075175
BC00718=46382,989307,1075175
BC00719=42015,987930,1075175
BC00720=86350,984014,1075175
BC00721=118186,882849,1075175
BC00722=118313,879045,1075175
BC00723=118363,877523,1075175
BC00724=127351,877496,1075175
BC00725=127300,879018,1075175
BC00726=127173,882822,1075175
BC00727=149531,895732,1075175
BC00728=148249,891267,1075175
BC00729=148034,889482,1075175
BC00730=151775,889498,1075175
BC00731=152288,891284,1075175
BC00732=153569,895750,1075175
BC00733=119302,902119,1075175
BC00734=119440,897649,1075175
BC00735=119495,895861,1075175
BC00736=115974,895890,1075175
BC00737=115919,897678,1075175
BC00738=115781,902148,1075175
BC00739=206850,915693,1075175
BC00740=246637,921611,1075175
BC00741=251241,924622,1075175
BC00742=253082,925827,1075175
BC00743=305626,902567,1075175
BC00744=289523,905356,1075175
BC00745=289523,905356,1075175
BC00746=289382,905334,1075175
BC00747=289381,905334,1075175
BC00748=265782,900020,1075175
BC00749=265246,895833,1075175
BC00750=152805,918674,1075175
BC00751=155644,922700,1075175
BC00752=156780,924310,1075175
BC00753=187141,913105,1075175
BC00754=182251,913961,1075175
BC00755=179648,914418,1075175
BC00756=179441,914454,1075175
BC00757=120688,931609,1075175
BC00758=120688,931609,1036122
BC00759=120688,931609,1036122
BC00760=135499,922155,1075175
BC00761=196755,924293,1075175
BC00762=204603,922909,1075175
BC00763=210067,918954,1075175
BC00764=285493,836258,1075175
BC00765=322674,778579,1075175
BC00766=322674,778579,1075175
BC00767=322674,778579,1075175
BC00768=322674,778579,1075175
BC00769=322674,778579,1075175
BC00770=322674,778579,1075175
BC00771=322674,778579,1075175
BC00772=322674,778579,1075175
BC00773=272555,769164,1075175
BC00774=266479,768023,1075175
BC00775=266479,768023,1075175
BC00776=267479,770239,1071365
BC00777=266799,769335,1075175
BC00778=266479,768023,1075175
BC00779=266479,768023,1075175
BC00780=266479,768023,1075175
BC00781=266479,768023,1075175
BC00782=235984,786404,1075175
BC00783=235984,786404,1075175
BC00784=235984,786404,1075175
BC00785=235984,786404,1075175
BC00786=235984,786404,1075175
BC00787=235984,786404,1075175
BC00788=235984,786404,1075175
BC00789=235984,786404,1075175
BC00790=237203,787368,1075175
BC00791=295022,827394,1075175
BC00792=205701,931185,1075175
BC00793=204812,932218,1075175
BC00794=205671,937629,1075175
BC00795=206015,939793,1075175
BC00796=202546,941762,1075175
BC00797=218293,952795,1075175
BC00798=218466,950486,1075175
BC00799=218898,944716,1075175
BC00800=188226,925402,1075175
BC00801=189298,932104,1075175
BC00802=189728,934784,1075175
BC00803=185375,937227,1075175
BC00804=184946,934546,1075175
BC00805=183874,927845,1075175
BC00806=163256,940528,1075175
BC00807=166760,944877,1075175
BC00808=168161,946617,1075175
BC00809=172960,943924,1075175
BC00810=171559,942185,1075175
BC00811=168055,937836,1075175
BC00812=205604,952176,1075175
BC00813=237375,964309,1075175
BC00814=234858,970014,1075175
BC00815=233851,972296,1075175
BC00816=237408,970622,1075175
BC00817=238426,968449,1075175
BC00818=241139,962660,1075175
BC00819=186195,958850,1075175
BC00820=137530,955476,1075175
BC00821=142340,959691,1075175
BC00822=135217,966057,1075175
BC00823=135217,966057,1075175
BC00824=134381,966543,1075175
BC00825=132263,964948,1075175
BC00826=126968,960962,1075175
BC00827=137530,955476,1075175
BC00828=284870,850327,1075175
BC00829=323104,941595,1075175
BC00830=323297,942087,1075175
BC00831=323297,942087,1075175
BC00832=323297,942087,1075175
BC00833=324969,946346,1075175
BC00834=377020,937331,1075175
BC00835=379859,936839,1075175
BC00836=379326,935482,1075175
BC00837=377994,932088,1075175
BC00838=387025,925803,1075175
BC00839=391871,922431,1075175
BC00840=387133,926188,1075175
BC00841=385238,927691,1075175
BC00842=381091,925537,1075175
BC00843=365308,912570,1075175
BC00844=363166,908743,1075175
BC00845=364796,906869,1075175
BC00846=368870,902183,1075175
BC00847=358157,902408,1075175
BC00848=354876,908652,1075175
BC00849=353564,911150,1075175
BC00850=349138,907302,1075175
BC00851=357572,916934,1075175
BC00852=359178,914754,1075175
BC00853=363193,909304,1075175
BC00854=322758,853588,1075175
BC00855=135439,955204,1075175
BC00856=139952,957848,1075175
BC00857=141757,958906,1075175
BC00858=133040,997822,1075175
BC00859=133065,977483,1075175
BC00860=144047,1040883,1075175
BC00861=142698,1043050,1075175
BC00862=139327,1048468,1075175
BC00863=139327,1048468,1075175
BC00864=95619,955204,1075175
BC00865=100132,965528,1075175
BC00866=101937,966586,1075175
BC00867=93220,1005502,1075175
BC00868=93220,1005502,1075175
BC00869=93221,1030527,1075216
BC00870=93221,1030527,1075216
BC00871=99566,1045795,1075190
BC00872=142698,1043050,1075175
BC00873=206177,1018673,1075175
BC00874=252443,1048931,1075175
BC00875=258757,1029159,1075175
BC00876=290253,930536,1075175
BC00877=290253,930536,1075175
BC00878=290253,930536,1075175
BC00879=297151,966120,1075172
BC00880=297151,997903,1075172
BC00881=297151,997903,1075172
BC00882=297194,1021413,1075172
BC00883=297194,1021413,1075172
BC00884=21214,672831,1075175
BC00885=21214,672831,429902
BC00886=66815,724118,419761
BC00887=110240,772957,337669
BC00888=124996,789553,122283
BC00889=124996,789553,122283
BC00890=124996,789553,122283
BC00891=124996,789553,122283
BC00892=124996,789553,122283
BC00893=124996,789553,122283
BC00894=124996,789553,122283
BC00895=124996,789553,122283
BC00896=124996,789553,122283
BC00897=124996,789553,122283
BC00898=136729,789553,283981
BC00899=136729,789553,283981
BC00900=136729,789553,283981
BC00901=136729,789553,283981
BC00902=136729,789553,283981
BC00903=136729,789553,283981
BC00904=136729,789553,283981
BC00905=136729,789553,283981
BC00906=136729,789553,283981
BC00907=136729,789553,283981
BC00908=163194,789553,386705
BC00909=163194,789553,386705
BC00910=163194,789553,386705
BC00911=163194,789553,386705
BC00912=163194,789553,386705
BC00913=163194,789553,386705
BC00914=163194,789553,386705
BC00915=163194,789553,386705
BC00916=163194,789553,386705
BC00917=163194,789553,386705
BC00918=110240,772957,337669
BC00919=66815,724118,419761
BC00920=66815,670858,419761
BC00921=252765,670858,277331
BC00922=322808,760288,131711
BC00923=322808,760288,131711
BC00924=322808,760288,131711
BC00925=322808,760288,131711
BC00926=322808,760288,131711
BC00927=322808,760288,131711
BC00928=322808,760288,131711
BC00929=322808,760288,131711
BC00930=322808,760288,131711
BC00931=335534,789553,204922
BC00932=335534,789553,204922
BC00933=335534,789553,204922
BC00934=335534,789553,204922
BC00935=335534,789553,204922
BC00936=335534,789553,204922
BC00937=335534,789553,204922
BC00938=335534,789553,204922
BC00939=335534,789553,204922
BC00940=344006,752651,139062
BC00941=344006,752651,139062
BC00942=344006,752651,139062
BC00943=344006,752651,139062
BC00944=344006,752651,139062
BC00945=344006,752651,139062
BC00946=344006,752651,139062
BC00947=344006,752651,139062
BC00948=344006,752651,139062
BC00949=300933,750795,218908
BC00950=283893,750061,250495
BC00951=276320,749735,264534
BC00952=276320,749735,264534
BC00953=276320,749735,264534
BC00954=276320,749735,264534
BC00955=276320,749735,264534
BC00956=276320,749735,264534
BC00957=276320,749735,264534
BC00958=276320,749735,264534
BC00959=276320,749735,264534
BC00960=248857,763770,138691
BC00961=248857,763770,138691
BC00962=248857,763770,138691
BC00963=248857,763770,138691
BC00964=248857,763770,138691
BC00965=248857,763770,138691
BC00966=248857,763770,138691
BC00967=248857,763770,138691
BC00968=248857,763770,138691
BC00969=287864,789553,132710
BC00970=287864,789553,132710
BC00971=287864,789553,132710
BC00972=287864,789553,132710
BC00973=287864,789553,132710
BC00974=287864,789553,132710
BC00975=287864,789553,132710
BC00976=287864,789553,132710
BC00977=287864,789553,132710
BC00978=287864,789553,132710
BC00979=287864,789553,132710
BC00980=287864,789553,132710
BC00981=279829,789553,53
BC00982=279829,789553,53
BC00983=279829,789553,53
BC00984=279829,789553,53
BC00985=279829,789553,53
BC00986=279829,789553,53
BC00987=279829,789553,53
BC00988=279829,789553,53
BC00989=279829,789553,53
BC00990=279829,789553,53
BC00991=279829,789553,53
BC00992=279829,789553,53
BC00993=279829,789553,53
BC00994=312324,789553,158805
BC00995=312324,789553,158805
BC00996=312324,789553,158804
BC00997=312324,789553,158805
BC00998=312324,789553,158805
BC00999=312324,789553,158805
BC01000=303082,768394,105099
BC01001=303082,768394,105099
BC01002=303082,768394,105099
BC01003=303082,768394,105099
BC01004=303082,768394,105099
BC01005=303082,768394,105099
BC01006=287868,781442,183325
BC01007=278410,789553,231953
BC01008=278410,789553,231953
BC01009=278410,789553,231953
BC01010=278410,789553,231953
BC01011=278410,789553,231953
BC01012=278410,789553,231953
BC01013=283893,750061,250495
BC01014=300933,750795,218908
BC01015=376723,772526,120737
BC01016=376723,772526,120737
BC01017=376723,772526,120737
BC01018=376723,772526,120737
BC01019=376723,772526,120737
BC01020=376723,772526,120737
BC01021=385013,737075,95404
BC01022=385013,737075,95404
BC01023=385013,737075,95404
BC01024=385013,737075,95404
BC01025=385013,737075,95404
BC01026=385013,737075,95404
BC01027=365962,760163,122379
BC01028=365962,760163,122379
BC01029=365962,760163,122379
BC01030=365962,760163,122379
BC01031=365962,760163,122379
BC01032=365962,760163,122379
BC01033=365962,760163,122379
BC01034=252765,670858,277331
BC01035=66815,670858,419761
BC01036=66815,724118,419761
BC01037=110240,772957,337669
BC01038=118803,789553,240458
BC01039=118803,789553,240458
BC01040=118803,789553,240458
BC01041=118803,789553,240458
BC01042=118803,789553,240458
BC01043=118803,789553,240458
BC01044=130259,789553,198376
BC01045=110709,789553,198376
BC01046=113251,789553,198376
BC01047=113251,789553,198376
BC01048=113251,789553,198376
BC01049=113251,789553,198376
BC01050=113251,789553,198376
BC01051=113251,789553,198376
BC01052=113251,789553,198376
BC01053=113251,789553,198376
BC01054=113251,789553,198376
BC01055=113251,789553,198376
BC01056=113251,789553,198376
BC01057=113251,789553,198376
BC01058=113251,789553,198376
BC01059=113251,789553,228042
BC01060=113251,789553,280292
BC01061=113251,789553,280290
BC01062=113251,789553,280290
BC01063=113251,789553,280290
BC01064=113251,789553,280290
BC01065=113251,789553,280290
BC01066=113251,789553,280290
BC01067=113251,789553,280290
BC01068=110240,772957,337669
BC01069=66815,724118,419761
BC01070=66815,670858,419761
BC01071=252765,670858,277331
BC01072=298333,782774,240815
BC01073=298333,782774,240815
BC01074=298333,782774,240815
BC01075=298333,782774,240815
BC01076=298333,782774,240815
BC01077=298333,782774,240815
BC01078=277596,773081,190929
BC01079=277596,773081,190929
BC01080=277596,773081,190929
BC01081=277596,773081,190929
BC01082=277596,773081,190929
BC01083=277596,773081,190929
BC01084=252765,670858,277331
BC01085=66815,670858,419761
BC01086=66815,724118,419761
BC01087=110240,772957,337669
BC01088=116545,789553,319269
BC01089=116545,789553,319269
BC01090=116545,789553,319269
BC01091=116545,789553,319269
BC01092=116545,789553,319269
BC01093=116545,789553,319269
BC01094=104258,789553,379308
BC01095=104258,789553,379308
BC01096=104258,789553,379308
BC01097=104258,789553,379308
BC01098=104258,789553,379308
BC01099=104258,789553,379308
BC01100=110240,772957,337669
BC01101=66815,724118,419761
BC01102=66815,670858,419761
BC01103=252765,670858,277331
BC01104=286674,787255,240962
BC01105=286675,787255,240962
BC01106=286675,787255,240962
BC01107=286675,787255,240962
BC01108=286674,787255,240962
BC01109=286674,787255,240962
BC01110=267109,758037,158941
BC01111=267109,758037,158941
BC01112=267109,758037,158941
BC01113=267109,758037,158941
BC01114=267109,758037,158941
BC01115=267109,758037,158941
BC01116=283893,750061,250495
BC01117=360336,760725,110934
BC01118=360336,760725,110934
BC01119=360336,760725,110934
BC01120=360336,760725,110934
BC01121=360336,760725,110934
BC01122=360336,760725,110934
BC01123=371149,789553,191296
BC01124=371149,789553,191296
BC01125=371149,789553,191296
BC01126=371149,789553,191296
BC01127=371149,789553,191296
BC01128=371149,789553,191296
BC01129=283893,750061,250495
BC01130=292970,789553,136523
BC01131=292970,789553,136523
BC01132=292970,789553,136523
BC01133=292970,789553,136523
BC01134=292970,789553,136523
BC01135=292970,789552,136519
BC01136=292970,789553,136523
BC01137=292970,789553,136523
BC01138=256495,759418,21571
BC01139=256495,759418,21571
BC01140=256495,759418,21571
BC01141=256495,759418,21571
BC01142=256495,759418,21571
BC01143=256495,759418,21571
BC01144=256075,748610,41729
BC01145=255916,738170,60084
BC01146=255916,738170,60084
BC01147=255916,738170,60084
BC01148=255916,738170,60084
BC01149=255916,738170,60084
BC01150=255916,738170,60084
BC01151=262339,748900,193466
BC01152=165820,667836,534036
BC01153=21214,672831,1075175
EC00000=798156,1112951
EC00001=798156,1112951
EC00002=798156,1112951
EC00003=798156,1112951
EC00004=798156,1112951
EC00005=798156,1112951
EC00006=798156,1112951
EC00007=798156,1112951
EC00008=798156,1112951
EC00009=798156,1112951
EC00010=798156,1112951
EC00011=798156,1112951
EC00012=798156,1112951
EC00013=798156,1112951
EC00014=798156,1112951
EC00015=798156,1112951
EC00016=798156,1112951
EC00017=798156,1112951
EC00018=798156,1112951
EC00019=798156,1112951
EC00020=798156,1112951
EC00021=798156,1112951
EC00022=798156,1112951
EC00023=798156,1112951
EC00024=798156,1112951
EC00025=798156,1112951
EC00026=798156,1112951
EC00027=798156,1112951
EC00028=798156,1112951
EC00029=798156,1112951
EC00030=798156,1112951
EC00031=798156,1112951
EC00032=798156,1112951
EC00033=798156,1112951
EC00034=798156,1112951
EC00035=798156,1112951
EC00036=798156,1112951
EC00037=798156,1112951
EC00038=798156,1112951
EC00039=798156,1112951
EC00040=798156,1112951
EC00041=798155,1112950
EC00042=798155,1112950
EC00043=798155,1112950
EC00044=798154,1112949
EC00045=798154,1112949
EC00046=798154,1112949
EC00047=798154,1112949
EC00048=798154,1112949
EC00049=798153,1112949
EC00050=798156,1112951
EC00051=798156,1112951
EC00052=798156,1112951
EC00053=798156,1112951
EC00054=798156,1112951
EC00055=798156,1112951
EC00056=798156,1112951
EC00057=798156,1112951
EC00058=798156,1112951
EC00059=798156,1112951
EC00060=798156,1112951
EC00061=798156,1112951
EC00062=798156,1112951
EC00063=798156,1112951
EC00064=798156,1112951
EC00065=798156,1112951
EC00066=798156,1112951
EC00067=798156,1112951
EC00068=798156,1112951
EC00069=798156,1112951
EC00070=798155,1112950
EC00071=798155,1112950
EC00072=798156,1112951
EC00073=798156,1112951
EC00074=798156,1112951
EC00075=798156,1112951
EC00076=798156,1112951
EC00077=798156,1112951
EC00078=798156,1112951
EC00079=798156,1112951
EC00080=798156,1112951
EC00081=798156,1112951
EC00082=798156,1112951
EC00083=798156,1112951
EC00084=798156,1112951
EC00085=798156,1112951
EC00086=798156,1112951
EC00087=798156,1112951
EC00088=798156,1112951
EC00089=798156,1112951
EC00090=798156,1112951
EC00091=798156,1112951
EC00092=798156,1112951
EC00093=798156,1112951
EC00094=798156,1112951
EC00095=798156,1112951
EC00096=798156,1112951
EC00097=798156,1112951
EC00098=798156,1112951
EC00099=798156,1112951
EC00100=798156,1112951
EC00101=798156,1112951
EC00102=798156,1112951
EC00103=798156,1112951
EC00104=798156,1112951
EC00105=798156,1112951
EC00106=798156,1112951
EC00107=798156,1112951
EC00108=798156,1112951
EC00109=798156,1112951
EC00110=798156,1112951
EC00111=798156,1112951
EC00112=798156,1112951
EC00113=798156,1112951
EC00114=798156,1112951
EC00115=798156,1112951
EC00116=798156,1112951
EC00117=798156,1112951
EC00118=798156,1112951
EC00119=798156,1112951
EC00120=798156,1112951
EC00121=798156,1112951
EC00122=798156,1112951
EC00123=798156,1112951
EC00124=798156,1112951
EC00125=798156,1112951
EC00126=798156,1112951
EC00127=798156,1112951
EC00128=798156,1112951
EC00129=798156,1112951
EC00130=798156,1112951
EC00131=798156,1112951
EC00132=798156,1112951
EC00133=798156,1112951
EC00134=798156,1112951
EC00135=798156,1112951
EC00136=798156,1112951
EC00137=798156,1112951
EC00138=798156,1112951
EC00139=798156,1112951
EC00140=798156,1112951
EC00141=798156,1112951
EC00142=798156,1112951
EC00143=798156,1112951
EC00144=798156,1112951
EC00145=798156,1112951
EC00146=798156,1112951
EC00147=798156,1112951
EC00148=798156,1112951
EC00149=798156,1112951
EC00150=798156,1112951
EC00151=798156,1112951
EC00152=798156,1112951
EC00153=798156,1112951
EC00154=798156,1112951
EC00155=798156,1112951
EC00156=798156,1112951
EC00157=798156,1112951
EC00158=798156,1112951
EC00159=798156,1112951
EC00160=798156,1112951
EC00161=798156,1112951
EC00162=798156,1112951
EC00163=798156,1112951
EC00164=798156,1112951
EC00165=798156,1112951
EC00166=798156,1112951
EC00167=798156,1112951
EC00168=798156,1112951
EC00169=798156,1112951
EC00170=798156,1112951
EC00171=798156,1112951
EC00172=798156,1112951
EC00173=798156,1112951
EC00174=798156,1112951
EC00175=798156,1112951
EC00176=798156,1112951
EC00177=798156,1112951
EC00178=798156,1112951
EC00179=798156,1112951
EC00180=798155,1112950
EC00181=798155,1112950
EC00182=798155,1112950
EC00183=798155,1112950
EC00184=798155,1112950
EC00185=798155,1112950
EC00186=798155,1112950
EC00187=798155,1112950
EC00188=798155,1112950
EC00189=798155,1112950
EC00190=798155,1112950
EC00191=798155,1112950
EC00192=798156,1112951
EC00193=798156,1112951
EC00194=798156,1112951
EC00195=798156,1112951
EC00196=798156,1112951
EC00197=798156,1112951
EC00198=798156,1112951
EC00199=798155,1112950
EC00200=798155,1112950
EC00201=798155,1112950
EC00202=798155,1112950
EC00203=798155,1112950
EC00204=798155,1112950
EC00205=798155,1112950
EC00206=798155,1112950
EC00207=798155,1112950
EC00208=798155,1112950
EC00209=798156,1112951
EC00210=798156,1112951
EC00211=798156,1112951
EC00212=798156,1112951
EC00213=798156,1112951
EC00214=798156,1112951
EC00215=798156,1112951
EC00216=798156,1112951
EC00217=798156,1112951
EC00218=798156,1112951
EC00219=798156,1112951
EC00220=798156,1112951
EC00221=798156,1112951
EC00222=798156,1112951
EC00223=798156,1112951
EC00224=798155,1112950
EC00225=798155,1112950
EC00226=798155,1112950
EC00227=798155,1112950
EC00228=798155,1112950
EC00229=798155,1112950
EC00230=798155,1112950
EC00231=798155,1112950
EC00232=798155,1112950
EC00233=798155,1112950
EC00234=798155,1112950
EC00235=798155,1112950
EC00236=798156,1112951
EC00237=798156,1112951
EC00238=798156,1112951
EC00239=798156,1112951
EC00240=798156,1112951
EC00241=798156,1112951
EC00242=798156,1112951
EC00243=798155,1112950
EC00244=798155,1112950
EC00245=798155,1112950
EC00246=798155,1112950
EC00247=798155,1112950
EC00248=798155,1112950
EC00249=798155,1112950
EC00250=798155,1112950
EC00251=798155,1112950
EC00252=798155,1112950
EC00253=798156,1112951
EC00254=798156,1112951
EC00255=798155,1112950
EC00256=798156,1112951
EC00257=798156,1112951
EC00258=798156,1112951
EC00259=798156,1112951
EC00260=798156,1112951
EC00261=798156,1112951
EC00262=798156,1112951
EC00263=798156,1112951
EC00264=798156,1112951
EC00265=798156,1112951
EC00266=798156,1112951
EC00267=798156,1112951
EC00268=798156,1112951
EC00269=798156,1112951
EC00270=798156,1112951
EC00271=798156,1112951
EC00272=798156,1112951
EC00273=798156,1112951
EC00274=798156,1112951
EC00275=798156,1112951
EC00276=798156,1112951
EC00277=798156,1112951
EC00278=798156,1112951
EC00279=798156,1112951
EC00280=798156,1112951
EC00281=798156,1112951
EC00282=798156,1112951
EC00283=798156,1112951
EC00284=798156,1112951
EC00285=798156,1112951
EC00286=798156,1112951
EC00287=798156,1112951
EC00288=798156,1112951
EC00289=798156,1112951
EC00290=798156,1112951
EC00291=798156,1112951
EC00292=798156,1112951
EC00293=798156,1112951
EC00294=798156,1112951
EC00295=798156,1112951
EC00296=798156,1112951
EC00297=798156,1112951
EC00298=798156,1112951
EC00299=798156,1112951
EC00300=798155,1112950
EC00301=798154,1112950
EC00302=798154,1112950
EC00303=798154,1112950
EC00304=798154,1112950
EC00305=798154,1112950
EC00306=798154,1112950
EC00307=798154,1112950
EC00308=798155,1112950
EC00309=798155,1112950
EC00310=798155,1112950
EC00311=798155,1112950
EC00312=798155,1112950
EC00313=798155,1112950
EC00314=798155,1112950
EC00315=798155,1112950
EC00316=798156,1112951
EC00317=798156,1112951
EC00318=798156,1112951
EC00319=798156,1112951
EC00320=798156,1112951
EC00321=798156,1112951
EC00322=798156,1112951
EC00323=798156,1112951
EC00324=798156,1112951
EC00325=798156,1112951
EC00326=798156,1112951
EC00327=798156,1112951
EC00328=798156,1112951
EC00329=798156,1112951
EC00330=798156,1112951
EC00331=798156,1112951
EC00332=798156,1112951
EC00333=798156,1112951
EC00334=798156,1112951
EC00335=798156,1112951
EC00336=798156,1112951
EC00337=798156,1112951
EC00338=798156,1112951
EC00339=798156,1112951
EC00340=798156,1112951
EC00341=798156,1112951
EC00342=798156,1112951
EC00343=798156,1112951
EC00344=798156,1112951
EC00345=798156,1112951
EC00346=798156,1112951
EC00347=798156,1112951
EC00348=798156,1112951
EC00349=798156,1112951
EC00350=798155,1112950
EC00351=798155,1112950
EC00352=798155,1112950
EC00353=798155,1112950
EC00354=798155,1112950
EC00355=798155,1112950
EC00356=798155,1112950
EC00357=798155,1112950
EC00358=798155,1112950
EC00359=798155,1112950
EC00360=798156,1112951
EC00361=798156,1112951
EC00362=798156,1112951
EC00363=798156,1112951
EC00364=798156,1112951
EC00365=798156,1112951
EC00366=798156,1112951
EC00367=798156,1112951
EC00368=798156,1112951
EC00369=798156,1112951
EC00370=798156,1112951
EC00371=798156,1112951
EC00372=798156,1112951
EC00373=798156,1112951
EC00374=798156,1112951
EC00375=798156,1112951
EC00376=798156,1112951
EC00377=798156,1112951
EC00378=798156,1112951
EC00379=798156,1112951
EC00380=798156,1112951
EC00381=798156,1112951
EC00382=798156,1112951
EC00383=798156,1112951
EC00384=798156,1112951
EC00385=798156,1112951
EC00386=798155,1112951
EC00387=798156,1112951
EC00388=798156,1112951
EC00389=798156,1112951
EC00390=798156,1112951
EC00391=798156,1112951
EC00392=798156,1112951
EC00393=798156,1112951
EC00394=798156,1112951
EC00395=798156,1112951
EC00396=798156,1112951
EC00397=798156,1112951
EC00398=798156,1112951
EC00399=798156,1112951
EC00400=798156,1112951
EC00401=798156,1112951
EC00402=798156,1112951
EC00403=798156,1112951
EC00404=798156,1112951
EC00405=798156,1112951
EC00406=798156,1112951
EC00407=798156,1112951
EC00408=798156,1112951
EC00409=798156,1112951
EC00410=798156,1112951
EC00411=798156,1112951
EC00412=798156,1112951
EC00413=798156,1112951
EC00414=798156,1112951
EC00415=798156,1112951
EC00416=798156,1112951
EC00417=798156,1112951
EC00418=798156,1112951
EC00419=798156,1112951
EC00420=798156,1112951
EC00421=798156,1112951
EC00422=798156,1112951
EC00423=798156,1112951
EC00424=798156,1112951
EC00425=798156,1112951
EC00426=798156,1112951
EC00427=798156,1112951
EC00428=798156,1112951
EC00429=798156,1112951
EC00430=798156,1112951
EC00431=798156,1112951
